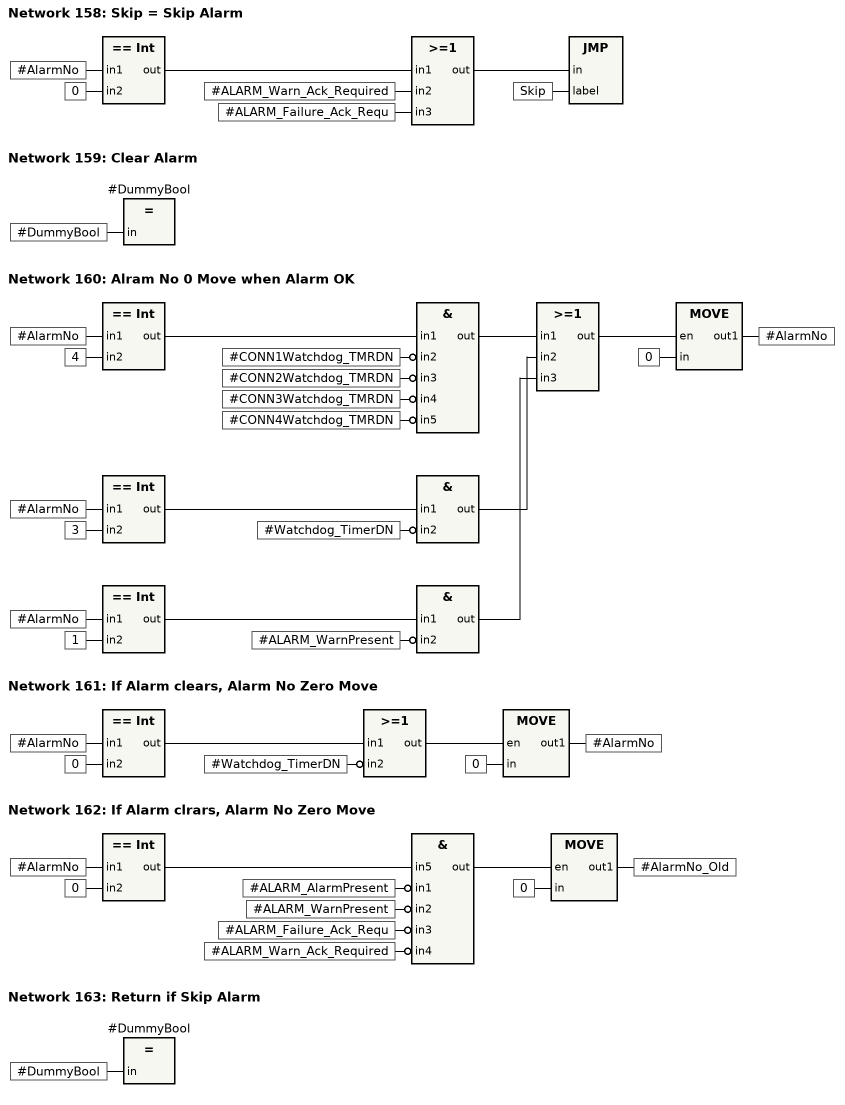
   IF (#AlarmNo = 0) OR #ALARM_Warn_Ack_Required OR #ALARM_Failure_Ack_Requ THEN GOTO Skip; END_IF;
END_REGION

REGION Network 159: Clear Alarm
   // >>>>>>>Clear Alarm>>>>>>>
   Clr:
   #DummyBool := #DummyBool;
END_REGION

REGION Network 160: Alram No 0 Move when Alarm OK
   IF ((#AlarmNo = 4) AND NOT #CONN1Watchdog_TMRDN AND NOT #CONN2Watchdog_TMRDN AND NOT #CONN3Watchdog_TMRDN AND NOT #CONN4Watchdog_TMRDN) OR ((#AlarmNo = 3) AND NOT #Watchdog_TimerDN) OR ((#AlarmNo = 1) AND NOT #ALARM_WarnPresent) THEN
       #AlarmNo := 0;
   END_IF;
END_REGION

REGION Network 161: If Alarm clears, Alarm No Zero Move
   IF (#AlarmNo = 0) OR NOT #Watchdog_TimerDN THEN #AlarmNo := 0; END_IF;
END_REGION

REGION Network 162: If Alarm clrars, Alarm No Zero Move
   IF (#AlarmNo = 0) AND NOT #ALARM_AlarmPresent AND NOT #ALARM_WarnPresent AND NOT #ALARM_Failure_Ack_Requ AND NOT #ALARM_Warn_Ack_Required THEN
       #AlarmNo_Old := 0;
   END_IF;
END_REGION

REGION Network 163: Return if Skip Alarm
   Skip:
   #DummyBool := #DummyBool;
END_REGION

REGION Network 164: Bit 16-19: Mode
   // 0 = Auto
   // 1= Single Start
   // 2 = Manual
   // 3= Local
   // 4= Test Mode
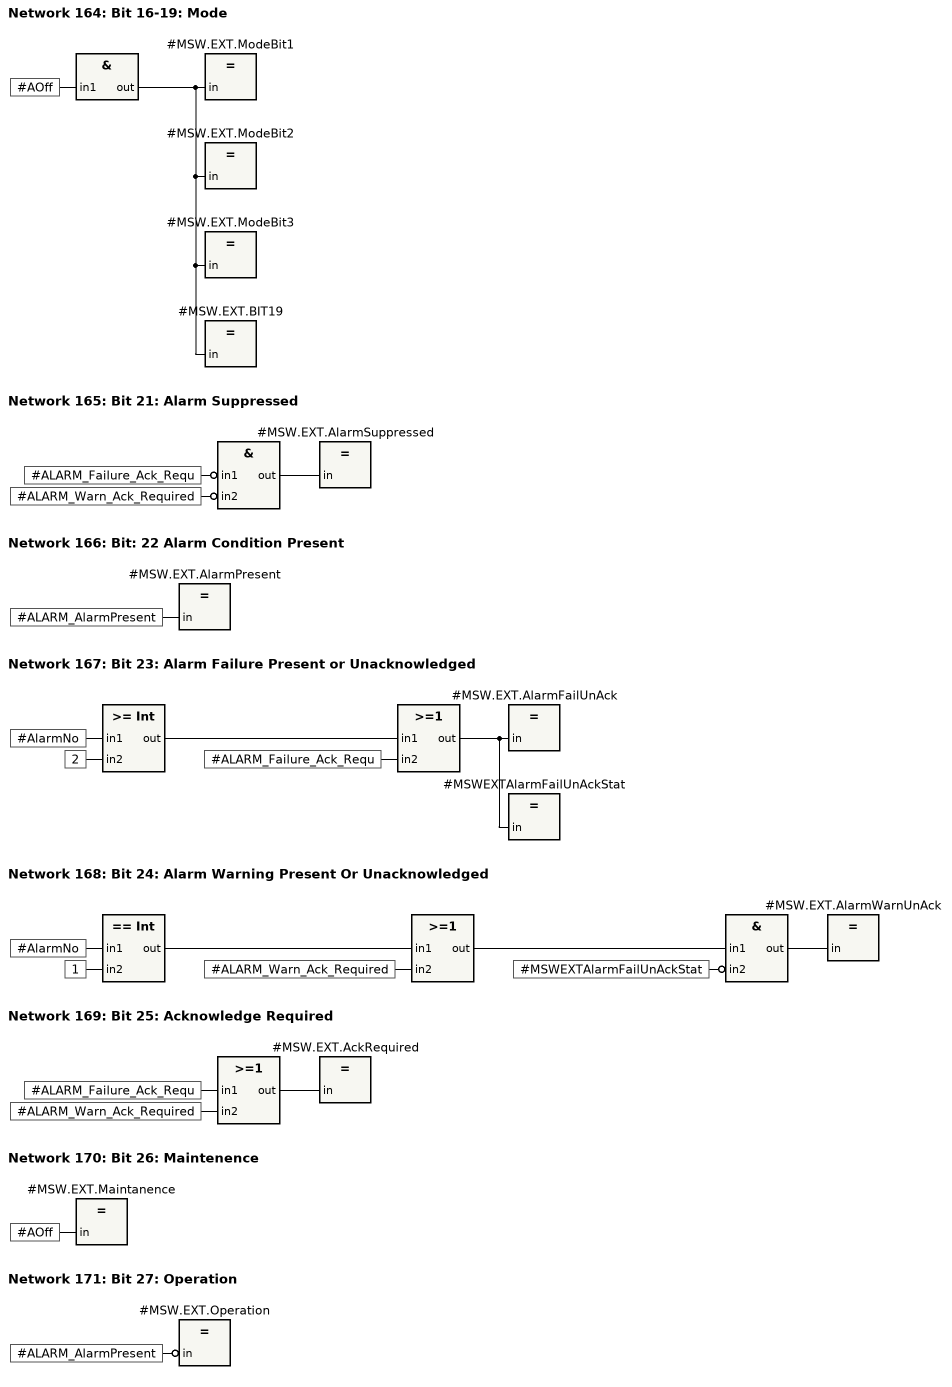
   #MSW.EXT.ModeBit1 := #AOff;
   #MSW.EXT.ModeBit2 := #AOff;
   #MSW.EXT.ModeBit3 := #AOff;
   #MSW.EXT.BIT19 := #AOff;
END_REGION

REGION Network 165: Bit 21: Alarm Suppressed
   #MSW.EXT.AlarmSuppressed := NOT #ALARM_Failure_Ack_Requ AND NOT #ALARM_Warn_Ack_Required;
END_REGION

REGION Network 166: Bit: 22 Alarm Condition Present
   #MSW.EXT.AlarmPresent := #ALARM_AlarmPresent;
END_REGION

REGION Network 167: Bit 23: Alarm Failure Present or Unacknowledged
   #MSW.EXT.AlarmFailUnAck := (#AlarmNo >= 2) OR #ALARM_Failure_Ack_Requ;
   #MSWEXTAlarmFailUnAckStat := #MSW.EXT.AlarmFailUnAck;
END_REGION

REGION Network 168: Bit 24: Alarm Warning Present Or Unacknowledged
   #MSW.EXT.AlarmWarnUnAck := ((#AlarmNo = 1) OR #ALARM_Warn_Ack_Required) AND NOT #MSWEXTAlarmFailUnAckStat;
END_REGION

REGION Network 169: Bit 25: Acknowledge Required
   #MSW.EXT.AckRequired := #ALARM_Failure_Ack_Requ OR #ALARM_Warn_Ack_Required;
END_REGION

REGION Network 170: Bit 26: Maintenence
   #MSW.EXT.Maintanence := #AOff;
END_REGION

REGION Network 171: Bit 27: Operation
   #MSW.EXT.Operation := NOT #ALARM_AlarmPresent;
END_REGION

REGION Network 172: Bit 28: Forced
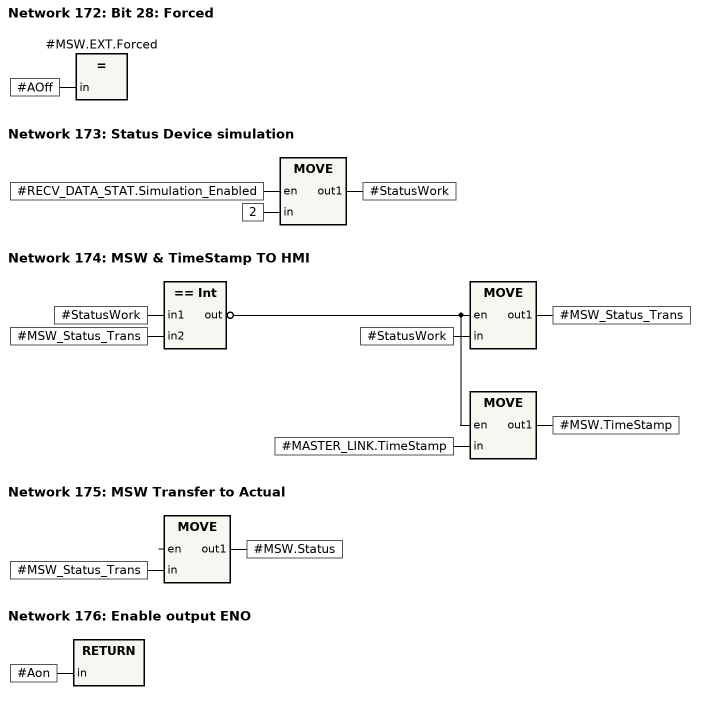
   #MSW.EXT.Forced := #AOff;
END_REGION

REGION Network 173: Status Device simulation
   IF #RECV_DATA_STAT.Simulation_Enabled THEN #StatusWork := 2; END_IF;
END_REGION

REGION Network 174: MSW & TimeStamp TO HMI
   #_w1 := NOT (#StatusWork = #MSW_Status_Trans);
   IF #_w1 THEN
       #MSW_Status_Trans := #StatusWork;
       #MSW.TimeStamp := #MASTER_LINK.TimeStamp;
   END_IF;
END_REGION

REGION Network 175: MSW Transfer to Actual
   #MSW.Status := #MSW_Status_Trans;
END_REGION

REGION Network 176: Enable output ENO
   IF #Aon THEN
       ENO := TRUE;
       RETURN;
   END_IF;
END_REGION
END_FUNCTION_BLOCK

FUNCTION_BLOCK "ACESYS_ISO_On_TCP_TSAP"   // FB228, FBD
TITLE = ACESYS V8.0 - Build 001 - ACESYS_ISO_On_TCP_TSAP
{ S7_Optimized_Access := 'FALSE' }
AUTHOR : FLSMIDTH
FAMILY : ACESYS
NAME : ISO_ON_TCP_TSAP
VERSION : 8.0
// Reference Block of ACESYS_SEND_RECV
   VAR_INPUT
      From_TCON_FC : Struct
         Connection_ID : Word;   // Valid from W#16#0001 to W#16#0FFF
         Connection_DEV_ID : Byte;   // B#16#01-IM151,#02-CPU31x,#03-S7319,#05-400CPU0,#15-400CPU1,#00-CP,10-CP(CPU1)
         Connection_ACT : Bool;   // ACTIVE=1; PASSIVE=0
         Connection_IP_ADDR1 : Int;   // Connection IP Address 1
         Connection_IP_ADDR2 : Int;   // Connection IP Address 2
         Connection_IP_ADDR3 : Int;   // Connection IP Address 3
         Connection_IP_ADDR4 : Int;   // Connection IP Address 4
         Connection_LOC_RS : Byte;   // Connection Local Rack/Slot
         Connection_CP_RS : Byte;   // Connection CP Rack/Slot
         Connection_REM_RS : Byte;   // Connection Remote Rack/Slot
         Connection_CONFIG_NO : Byte;   // B#16#01-CPU0NetA,#02CPU0NetB,#03CPU1NetA,#04CPU1NetB
      END_STRUCT;
   END_VAR
   VAR_OUTPUT
      TCON_PARM : TCON_IP_RFC;
   END_VAR
   VAR
      BlockInfo : Struct
         Ace_Version : Int;   // Acesys Block Version Number
         Ace_BuildNo : Int;   // Acesys Block Build Number
         DB_Number : Int;   // Block Instance DB Number
      END_STRUCT;
      SPECIFIED : Bool;
      DummyString : String[16];
      Connection_ID_Old : Word;
      Conn_String : String[16];
      TSAP16 : String[16];
      ID AT TSAP16 : Array[1..18] of Byte;
      Conn_EXT_HWID : GEOADDR;
   END_VAR
   VAR_TEMP
      Aon : Bool;
      DummyBool : Bool;
      DummyDWord : DWord;
      DummyInt : Int;
      DummyDInt : DInt;
      RET : Int;
      LOC_LEN : Int;
      REM_LEN : Int;
      TMP_INT : Int;
      LOC_RS : Int;
      TMP_RS : Int;
      TMP_DEV : Int;
      UDT_Length : Int;
      t_Zero : Int;
      Sample : Array[1..16] of Byte;
      b_Zero : Array[0..1] of Byte;
   END_VAR
   VAR_TEMP   // added for the SCL form of the ladder/FBD networks
      _w1 : Bool;
      _w2 : Bool;
      _w3 : Bool;
   END_VAR
BEGIN

REGION Network 1: Acesys Send Function Block based on Open Communication standard
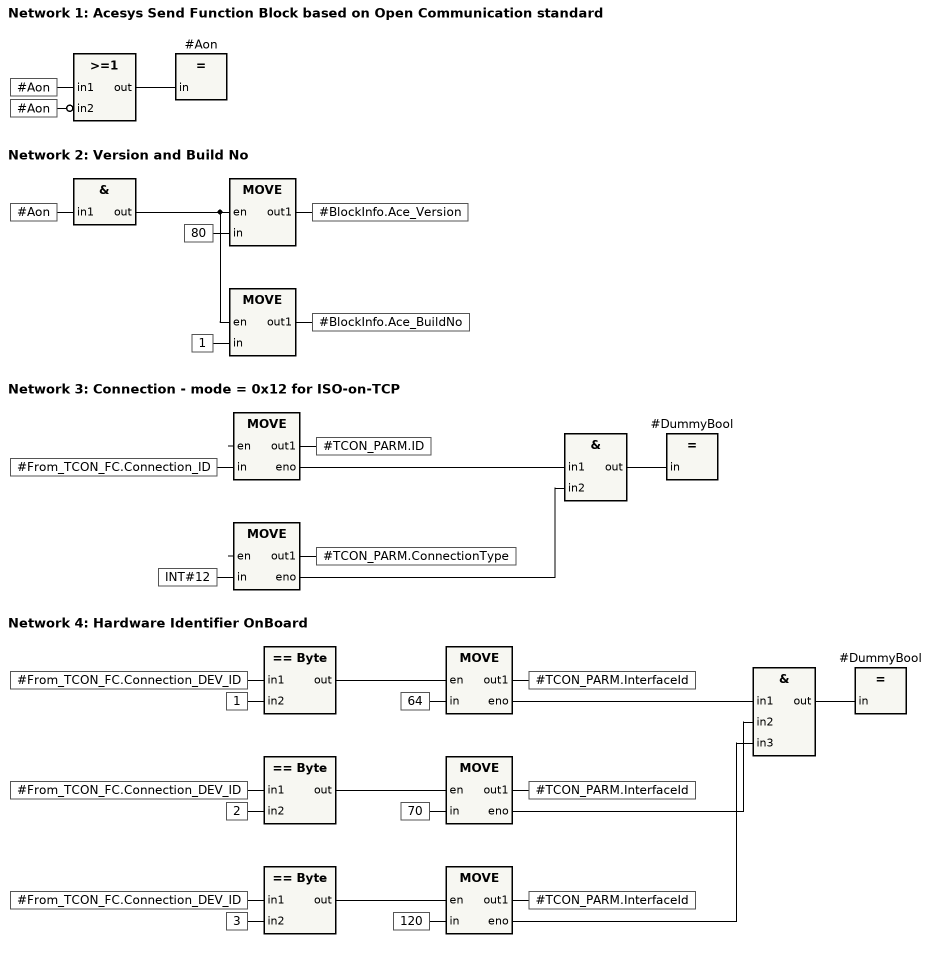
   #Aon := #Aon OR NOT #Aon;
END_REGION

REGION Network 2: Version and Build No
   IF #Aon THEN
       #BlockInfo.Ace_Version := 80;
       #BlockInfo.Ace_BuildNo := 1;
   END_IF;
END_REGION

REGION Network 3: Connection - mode = 0x12 for ISO-on-TCP
   // ENO of a box is taken as its EN; it also drops when the box reports an error
   #TCON_PARM.ID := #From_TCON_FC.Connection_ID;
   #TCON_PARM.ConnectionType := INT#12;
   #DummyBool := TRUE;
END_REGION

REGION Network 4: Hardware Identifier OnBoard
   #_w1 := #From_TCON_FC.Connection_DEV_ID = 1;
   IF #_w1 THEN #TCON_PARM.InterfaceId := 64; END_IF;
   #_w2 := #From_TCON_FC.Connection_DEV_ID = 2;
   IF #_w2 THEN #TCON_PARM.InterfaceId := 70; END_IF;
   #_w3 := #From_TCON_FC.Connection_DEV_ID = 3;
   IF #_w3 THEN #TCON_PARM.InterfaceId := 120; END_IF;
   #DummyBool := #_w1 AND #_w2 AND #_w3;
END_REGION

REGION Network 5: Hardware Identifier External
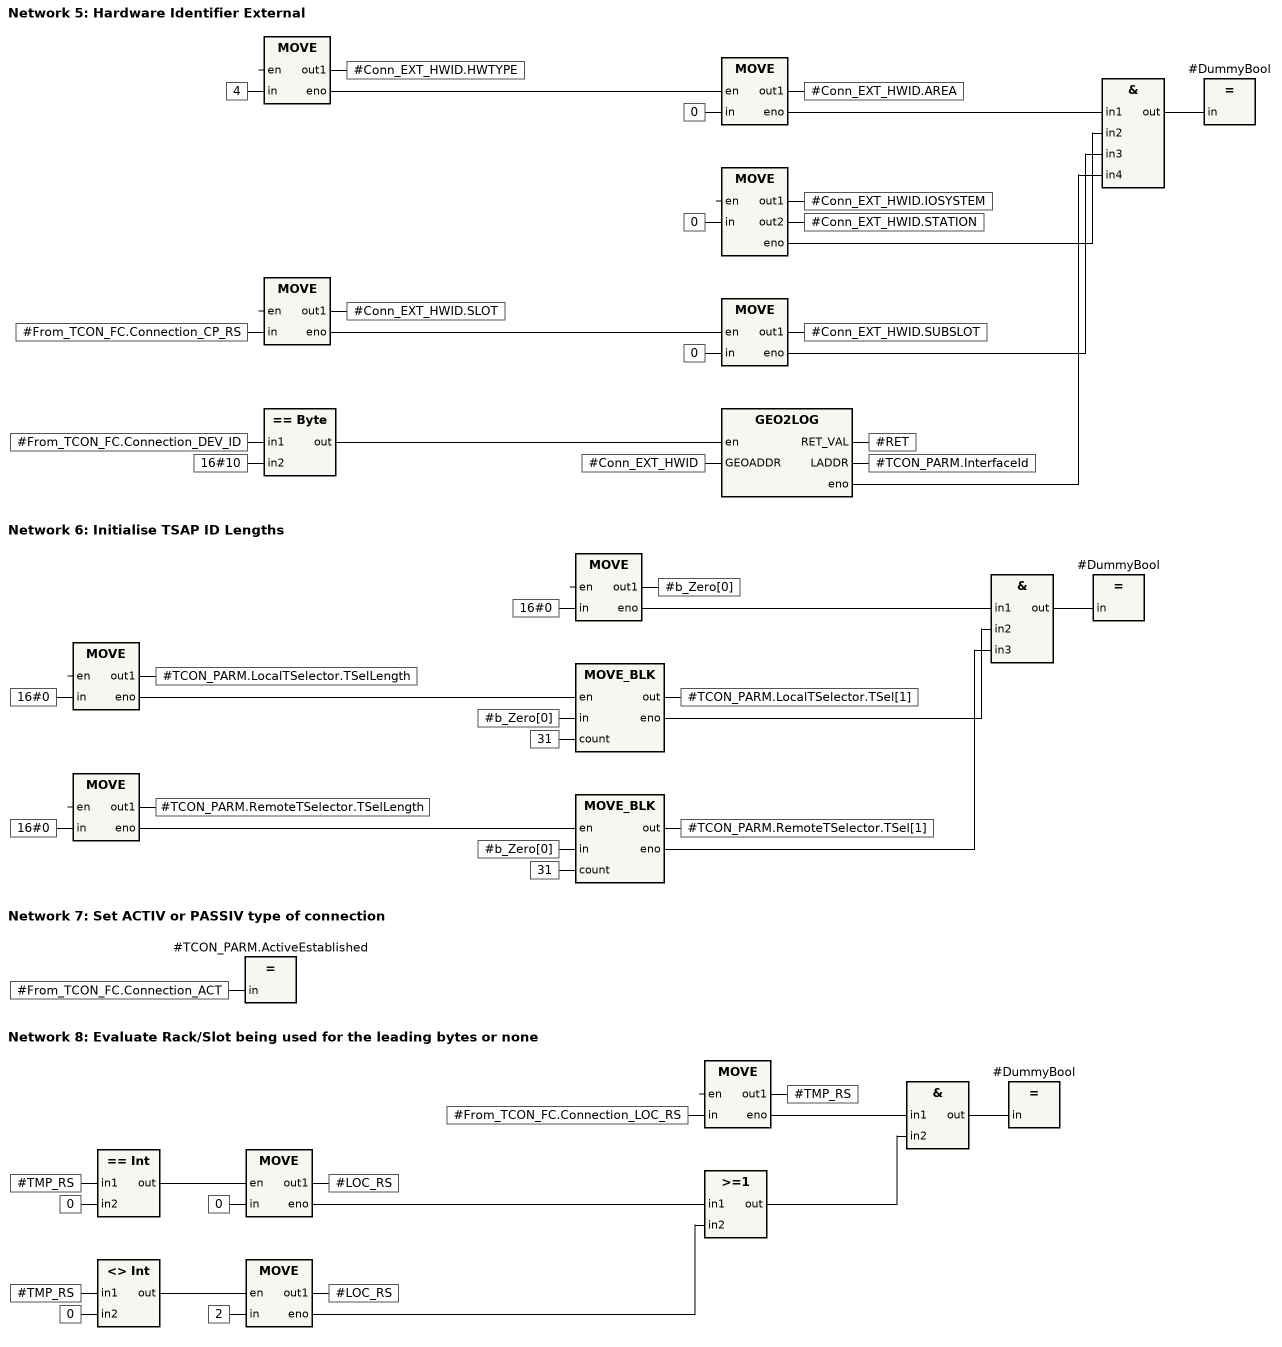
   // ENO of a box is taken as its EN; it also drops when the box reports an error
   #Conn_EXT_HWID.HWTYPE := 4;
   #Conn_EXT_HWID.AREA := 0;
   #Conn_EXT_HWID.IOSYSTEM := 0;
   #Conn_EXT_HWID.STATION := 0;
   #Conn_EXT_HWID.SLOT := #From_TCON_FC.Connection_CP_RS;
   #Conn_EXT_HWID.SUBSLOT := 0;
   #_w1 := #From_TCON_FC.Connection_DEV_ID = 16#10;
   IF #_w1 THEN #RET := GEO2LOG(GEOADDR := #Conn_EXT_HWID, LADDR => #TCON_PARM.InterfaceId); END_IF;
   #DummyBool := #_w1;
END_REGION

REGION Network 6: Initialise TSAP ID Lengths
   #b_Zero[0] := 16#0;
   #TCON_PARM.LocalTSelector.TSelLength := 16#0;
   MOVE_BLK(IN := #b_Zero[0], COUNT := 31, OUT => #TCON_PARM.LocalTSelector.TSel[1]);
   #TCON_PARM.RemoteTSelector.TSelLength := 16#0;
   MOVE_BLK(IN := #b_Zero[0], COUNT := 31, OUT => #TCON_PARM.RemoteTSelector.TSel[1]);
   #DummyBool := TRUE;
END_REGION

REGION Network 7: Set ACTIV or PASSIV type of connection
   // Receive Block Always Pasive
   #TCON_PARM.ActiveEstablished := #From_TCON_FC.Connection_ACT;
END_REGION

REGION Network 8: Evaluate Rack/Slot being used for the leading bytes or none
   // 1) If R/S = 0 ---> no leading bytes are requested.
   // 2) If R/S # 0 ---> two leading bytes are required.
   // ENO of a box is taken as its EN; it also drops when the box reports an error
   #TMP_RS := #From_TCON_FC.Connection_LOC_RS;
   #_w1 := #TMP_RS = 0;
   IF #_w1 THEN #LOC_RS := 0; END_IF;
   #_w2 := #TMP_RS <> 0;
   IF #_w2 THEN #LOC_RS := 2; END_IF;
   #DummyBool := #_w1 OR #_w2;
END_REGION

REGION Network 9: Check if ID is Changed
   // #MASTER_LINK.FIRST_SCAN - Removed
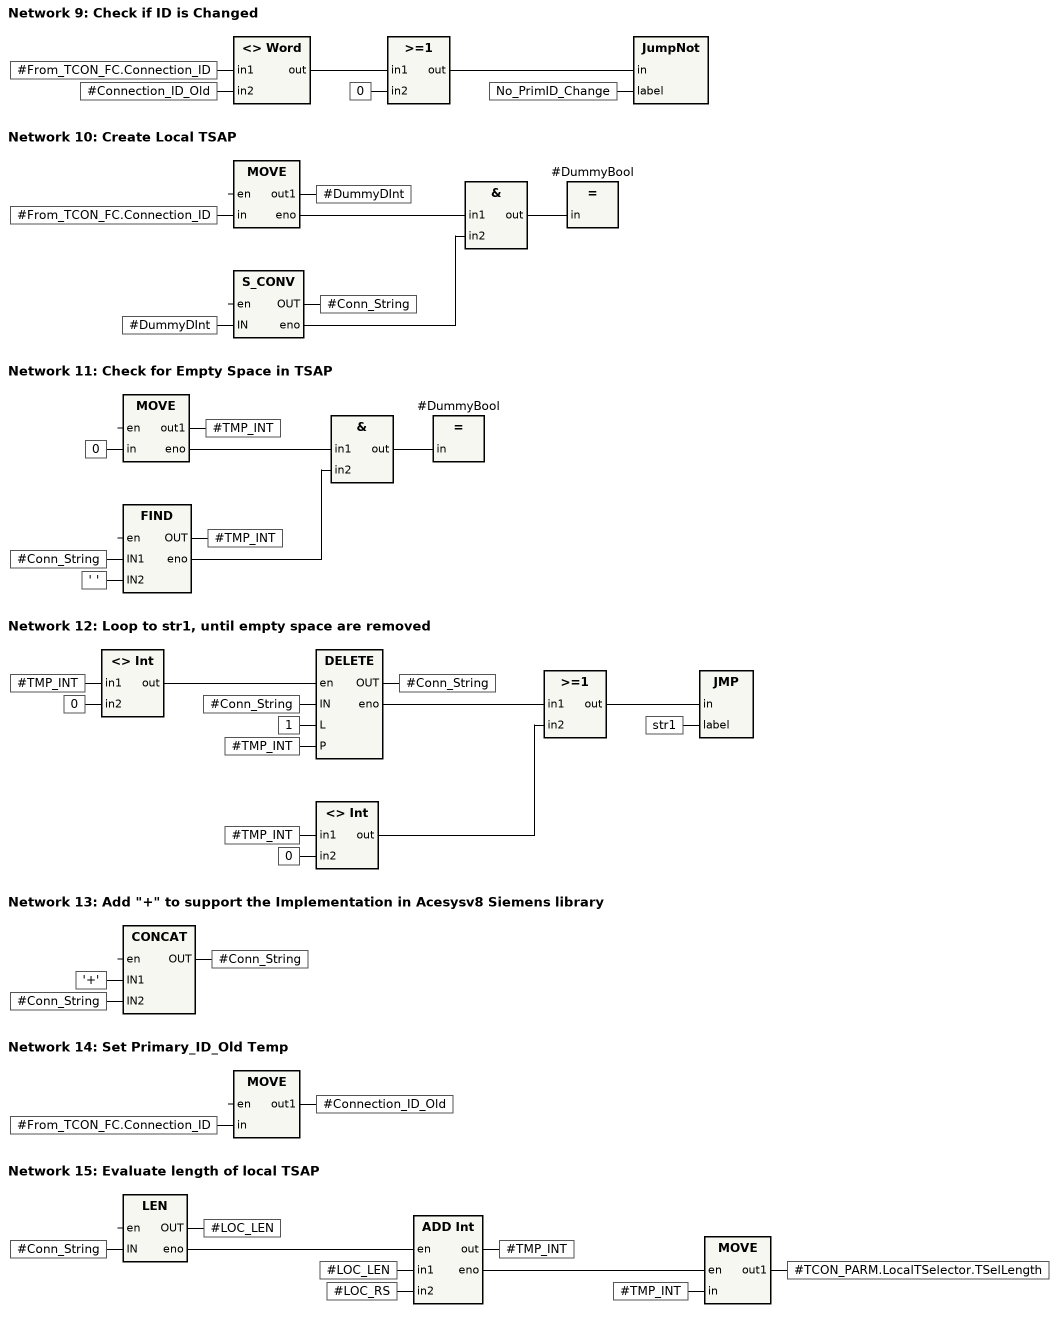
   // no SCL statement known for JumpNot: written as a call
   JumpNot(in := (#From_TCON_FC.Connection_ID <> #Connection_ID_Old) OR 0, label := No_PrimID_Change);
END_REGION

REGION Network 10: Create Local TSAP
   // Local TSAP = ID_Number
   // ENO of a box is taken as its EN; it also drops when the box reports an error
   #DummyDInt := #From_TCON_FC.Connection_ID;
   #Conn_String := S_CONV(IN := #DummyDInt);
   #DummyBool := TRUE;
END_REGION

REGION Network 11: Check for Empty Space in TSAP
   str1:
   #TMP_INT := 0;
   #TMP_INT := FIND(IN1 := #Conn_String, IN2 := ' ');
   #DummyBool := TRUE;
END_REGION

REGION Network 12: Loop to str1, until empty space are removed
   #_w1 := #TMP_INT <> 0;
   IF #_w1 THEN #Conn_String := DELETE(IN := #Conn_String, L := 1, P := #TMP_INT); END_IF;
   IF #_w1 OR (#TMP_INT <> 0) THEN GOTO str1; END_IF;
END_REGION

REGION Network 13: Add "+" to support the Implementation in Acesysv8 Siemens library
   #Conn_String := CONCAT(IN1 := '+', IN2 := #Conn_String);
END_REGION

REGION Network 14: Set Primary_ID_Old Temp
   No_PrimID_Change:
   #Connection_ID_Old := #From_TCON_FC.Connection_ID;
END_REGION

REGION Network 15: Evaluate length of local TSAP
   // #TSAP.LOC_TSAP
   // ENO of a box is taken as its EN; it also drops when the box reports an error
   #LOC_LEN := LEN(IN := #Conn_String);
   #TMP_INT := #LOC_LEN + #LOC_RS;
   #TCON_PARM.LocalTSelector.TSelLength := #TMP_INT;
END_REGION

REGION Network 16: copy local TSAP String to TSAP16 String!
   // #TSAP.LOC_TSAP
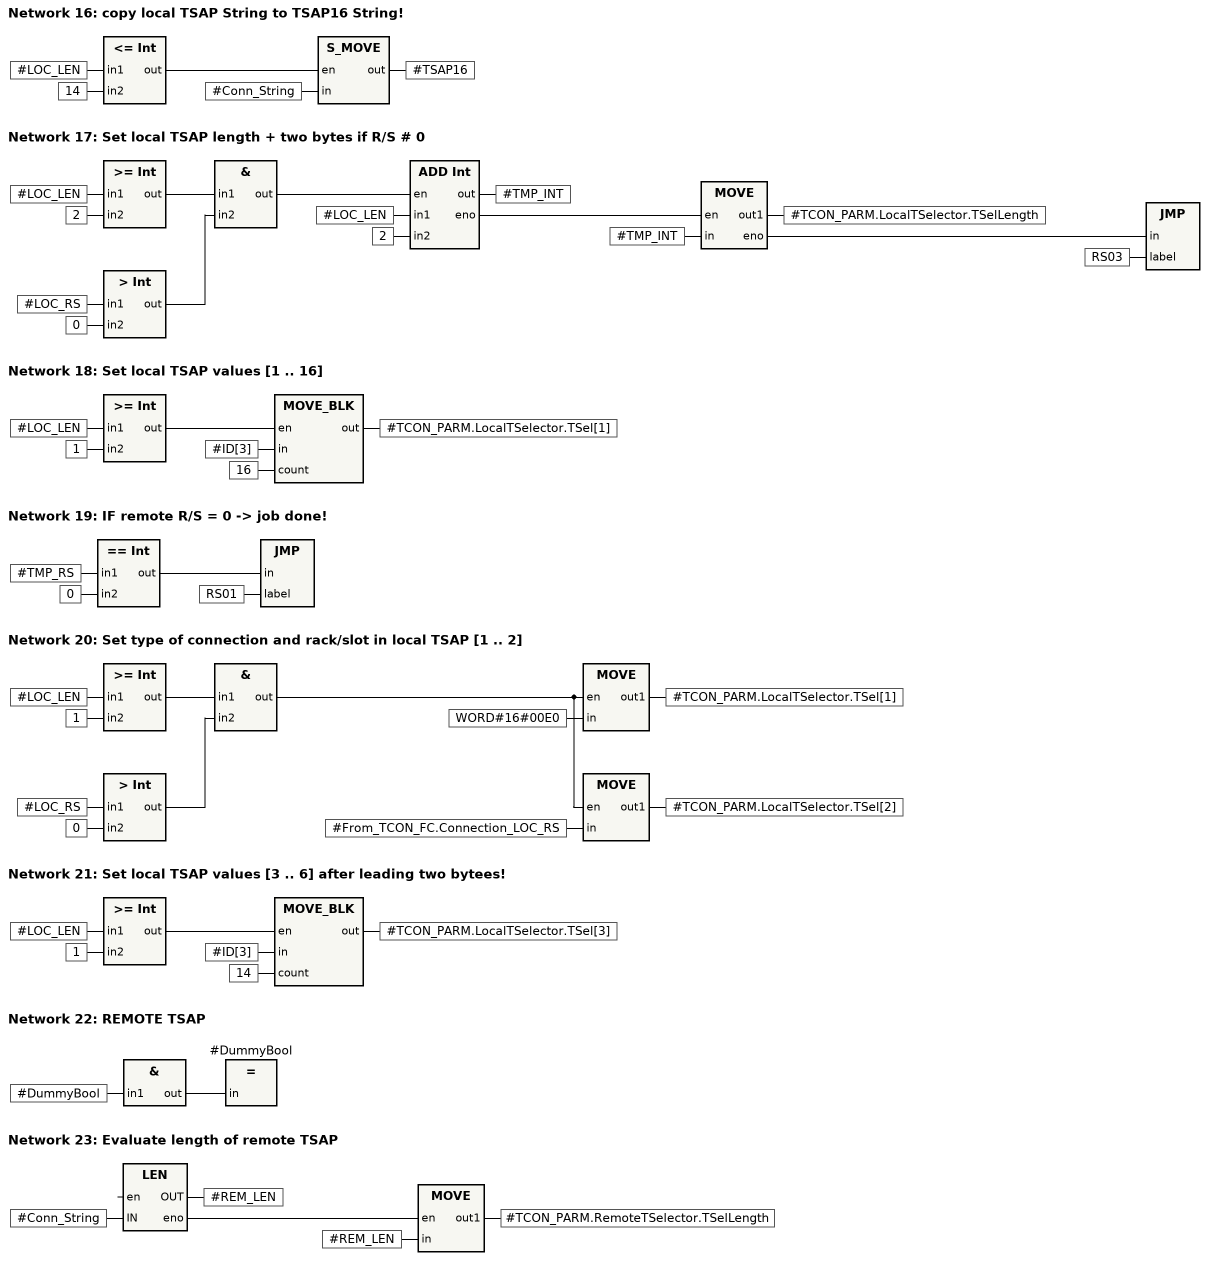
   IF #LOC_LEN <= 14 THEN #TSAP16 := #Conn_String; END_IF;
END_REGION

REGION Network 17: Set local TSAP length + two bytes if R/S # 0
   // ENO of a box is taken as its EN; it also drops when the box reports an error
   #_w1 := (#LOC_LEN >= 2) AND (#LOC_RS > 0);
   IF #_w1 THEN
       #TMP_INT := #LOC_LEN + 2;
       #TCON_PARM.LocalTSelector.TSelLength := #TMP_INT;
       GOTO RS03;
   END_IF;
END_REGION

REGION Network 18: Set local TSAP values [1 .. 16]
   // Fill in the entire local TSAP (without leading bytes)
   IF #LOC_LEN >= 1 THEN
       MOVE_BLK(IN := #ID[3], COUNT := 16, OUT => #TCON_PARM.LocalTSelector.TSel[1]);
   END_IF;
END_REGION

REGION Network 19: IF remote R/S = 0 -> job done!
   IF #TMP_RS = 0 THEN GOTO RS01; END_IF;
END_REGION

REGION Network 20: Set type of connection and rack/slot in local TSAP [1 .. 2]
   // B#16#E0 -> type of connection 
   // B#16#02 -> rack/slot of CPU
   RS03:
   IF (#LOC_LEN >= 1) AND (#LOC_RS > 0) THEN
       #TCON_PARM.LocalTSelector.TSel[1] := WORD#16#00E0;
       #TCON_PARM.LocalTSelector.TSel[2] := #From_TCON_FC.Connection_LOC_RS;
   END_IF;
END_REGION

REGION Network 21: Set local TSAP values [3 .. 6] after leading two bytees!
   IF #LOC_LEN >= 1 THEN
       MOVE_BLK(IN := #ID[3], COUNT := 14, OUT => #TCON_PARM.LocalTSelector.TSel[3]);
   END_IF;
END_REGION

REGION Network 22: REMOTE TSAP
   RS01:
   #DummyBool := #DummyBool;
END_REGION

REGION Network 23: Evaluate length of remote TSAP
   // Remote TSAP = Local TSAP (DummyString1)
   #REM_LEN := LEN(IN := #Conn_String);
   #TCON_PARM.RemoteTSelector.TSelLength := #REM_LEN;
END_REGION

REGION Network 24: copy remote TSAP String to TSAP16 String!
   // Remote TSAP = Local TSAP (DummyString)
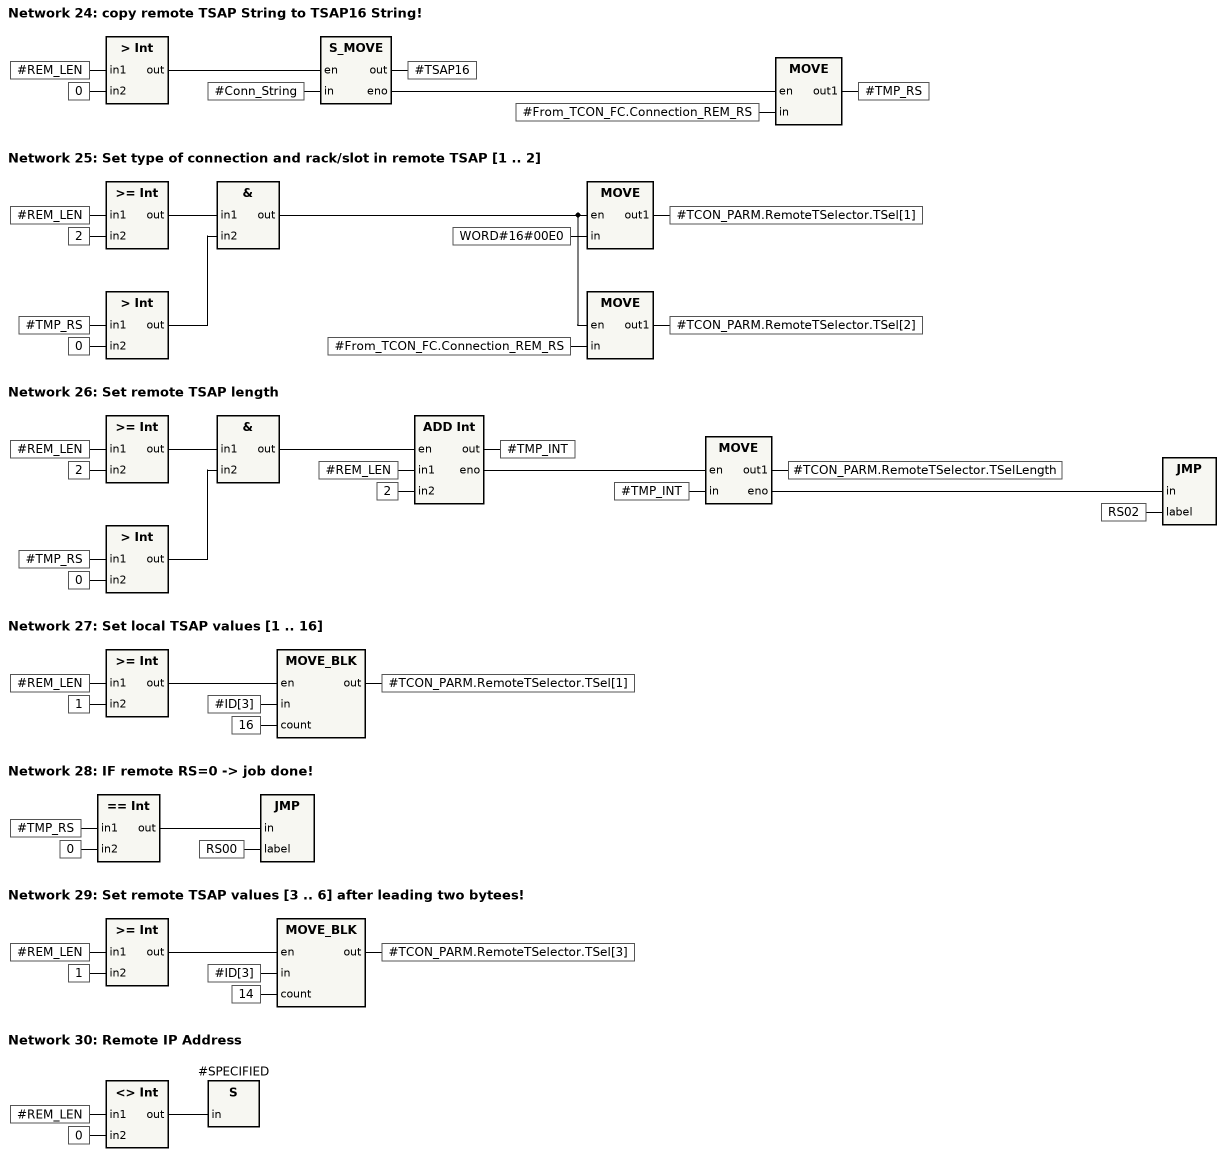
   IF #REM_LEN > 0 THEN
       #TSAP16 := #Conn_String;
       #TMP_RS := #From_TCON_FC.Connection_REM_RS;
   END_IF;
END_REGION

REGION Network 25: Set type of connection and rack/slot in remote TSAP [1 .. 2]
   // B#16#E0 -> type of connection 
   // B#16#02 -> rack/slot of CPU
   IF (#REM_LEN >= 2) AND (#TMP_RS > 0) THEN
       #TCON_PARM.RemoteTSelector.TSel[1] := WORD#16#00E0;
       #TCON_PARM.RemoteTSelector.TSel[2] := #From_TCON_FC.Connection_REM_RS;
   END_IF;
END_REGION

REGION Network 26: Set remote TSAP length
   // ENO of a box is taken as its EN; it also drops when the box reports an error
   #_w1 := (#REM_LEN >= 2) AND (#TMP_RS > 0);
   IF #_w1 THEN
       #TMP_INT := #REM_LEN + 2;
       #TCON_PARM.RemoteTSelector.TSelLength := #TMP_INT;
       GOTO RS02;
   END_IF;
END_REGION

REGION Network 27: Set local TSAP values [1 .. 16]
   // Fill in the entire local TSAP (without leading bytes)
   IF #REM_LEN >= 1 THEN
       MOVE_BLK(IN := #ID[3], COUNT := 16, OUT => #TCON_PARM.RemoteTSelector.TSel[1]);
   END_IF;
END_REGION

REGION Network 28: IF remote RS=0 -> job done!
   IF #TMP_RS = 0 THEN GOTO RS00; END_IF;
END_REGION

REGION Network 29: Set remote TSAP values [3 .. 6] after leading two bytees!
   RS02:
   IF #REM_LEN >= 1 THEN
       MOVE_BLK(IN := #ID[3], COUNT := 14, OUT => #TCON_PARM.RemoteTSelector.TSel[3]);
   END_IF;
END_REGION

REGION Network 30: Remote IP Address
   // Set length of the IP address if full-specified only !
   RS00:
   IF #REM_LEN <> 0 THEN #SPECIFIED := TRUE; END_IF;
END_REGION

REGION Network 31: Set not length of the IP address if unspecified !!!!
   // The remote IP address must be zero if
   // 1) remote TSAP is unspecified, or
   // 2) IP address is set up with zero!
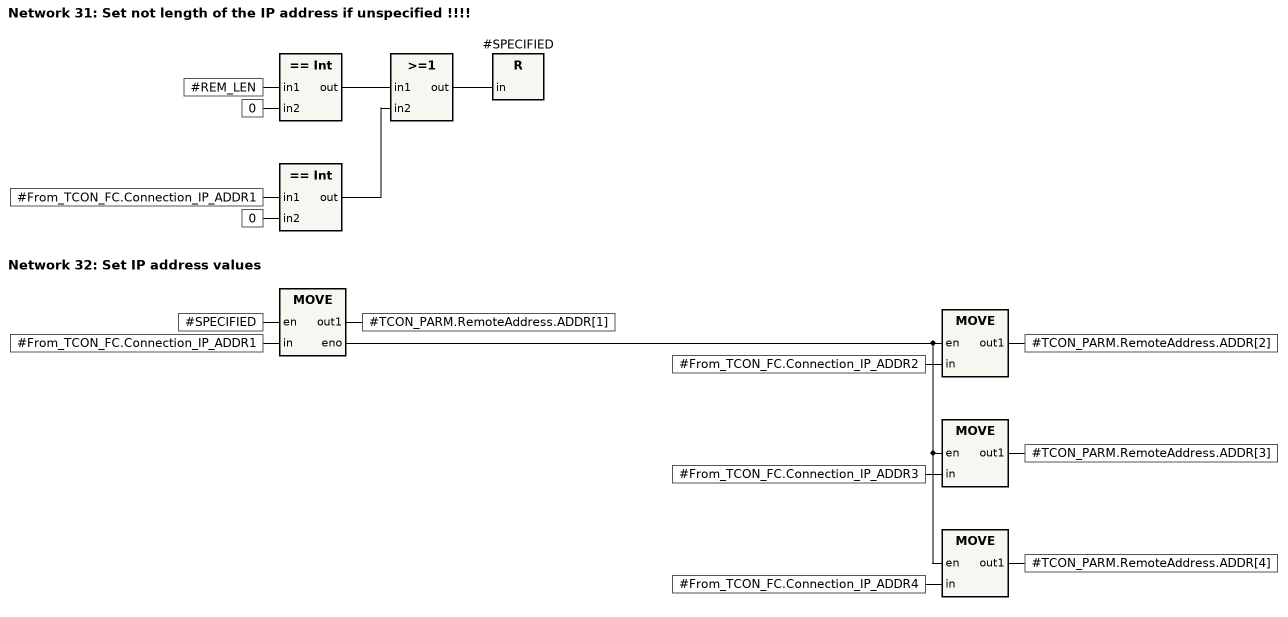
   IF (#REM_LEN = 0) OR (#From_TCON_FC.Connection_IP_ADDR1 = 0) THEN #SPECIFIED := FALSE; END_IF;
END_REGION

REGION Network 32: Set IP address values
   // ENO of a box is taken as its EN; it also drops when the box reports an error
   IF #SPECIFIED THEN
       #TCON_PARM.RemoteAddress.ADDR[1] := #From_TCON_FC.Connection_IP_ADDR1;
       #TCON_PARM.RemoteAddress.ADDR[2] := #From_TCON_FC.Connection_IP_ADDR2;
       #TCON_PARM.RemoteAddress.ADDR[3] := #From_TCON_FC.Connection_IP_ADDR3;
       #TCON_PARM.RemoteAddress.ADDR[4] := #From_TCON_FC.Connection_IP_ADDR4;
   END_IF;
END_REGION
END_FUNCTION_BLOCK

FUNCTION_BLOCK "ACESYS_PLC_DIAGV2"   // FB229, SCL
{ S7_Optimized_Access := 'FALSE' }
VERSION : 0.1
   VAR_INPUT
      HSBY_EN : Bool;   // Future Use
      OB33_ScanTime_In : Int;
      OB35_ScanTime_In : Int;
      CPU_Type : Int;   // Valid NO: "1200", "1500"
      Master_Link : "ACESYS_MASTER_LINK";
   END_VAR
   VAR_OUTPUT
      CPU_OK : Bool;   // CPU Status OK
      Type_Fault : Bool;   // CPU Type Fault
      CPUClock_Sec : USInt;
      CPUClock_Min : USInt;
      CPUClock_Hour : USInt;
      CPUClock_Day : USInt;
      CPUClock_Month : USInt;
      CPUClock_Year : UInt;
      OB01_ScanTime : Int;
      OB33_ScanTime : Int;
      OB35_ScanTime : Int;
      Memory_Total : DInt;
      Memory_Used : DInt;
      Mem_UsePercentage : Real;
      MSW : "ACESYS_HMI_STAT_32T";
   END_VAR
   VAR
      BlockInfo : Struct
         Ace_Version : Int;   // Acesys Block Version Number
         Ace_BuildNo : Int;   // Acesys Block Build Number
         DB_Number : Int;   // Block Instance DB Number
      END_STRUCT;
      FP_CMD : Struct   // Faceplate Commands
         Spare_08 : Bool;   // Bit8
         Spare_09 : Bool;   // Bit9
         Spare_10 : Bool;   // Bit10
         Spare_11 : Bool;   // Bit11
         Spare_12 : Bool;   // Bit12
         Spare_13 : Bool;   // Bit13
         Spare_14 : Bool;   // Bit14
         AckAlarm : Bool;   // Alarm Acknowledge
         Spare_00 : Bool;   // Bit0
         Spare_01 : Bool;   // Bit1
         Spare_02 : Bool;   // Bit2
         Spare_03 : Bool;   // Bit3
         Spare_04 : Bool;   // Bit4
         Spare_05 : Bool;   // Bit5
         Spare_06 : Bool;   // Bit6
         Spare_07 : Bool;   // Bit7
      END_STRUCT;
      FP_DIM : Struct
         Spare16 : Bool;
         Spare15 : Bool;
         Spare14 : Bool;
         Spare13 : Bool;
         Spare12 : Bool;
         Spare11 : Bool;
         Spare10 : Bool;
         Spare09 : Bool;
         Spare08 : Bool;
         Spare07 : Bool;
         Spare06 : Bool;
         Spare05 : Bool;
         Spare04 : Bool;
         Spare03 : Bool;
         Spare02 : Bool;
         Spare01 : Bool;
      END_STRUCT;
      FP_SHOW : Struct
         CPU_RUN_IND : Bool;
         Spare20 : Bool;
         Spare19 : Bool;
         Spare18 : Bool;
         Spare17 : Bool;
         Spare16 : Bool;
         Spare15 : Bool;
         Spare14 : Bool;
         Spare13 : Bool;
         Spare12 : Bool;
         Spare11 : Bool;
         CPU_MAINT : Bool;
         CPU_ERROR : Bool;
         OB1_ScanTime : Bool;
         OB33_ScanTime : Bool;
         OB35_ScanTime : Bool;
         Memory_Total : Bool;
         Memory_Used : Bool;
         Memory_Percent : Bool;
         Spare_10 : Bool;
         Spare_09 : Bool;
         Spare_08 : Bool;
         OB33ScanTimeIn : Bool;
         OB35ScanTimeIn : Bool;
         Spare_07 : Bool;
         Spare_06 : Bool;
         Spare_05 : Bool;
         Spare_04 : Bool;
         Spare_03 : Bool;
         Spare_02 : Bool;
         Spare_01 : Bool;
         Spare_00 : Bool;
      END_STRUCT;
      FP_PARM : Struct
         Spare16 : Bool;
         Spare15 : Bool;
         Spare14 : Bool;
         Spare13 : Bool;
         Spare12 : Bool;
         Spare11 : Bool;
         Spare10 : Bool;
         Spare09 : Bool;
         Spare08 : Bool;
         Spare07 : Bool;
         Spare06 : Bool;
         Spare05 : Bool;
         Spare04 : Bool;
         Spare03 : Bool;
         Spare02 : Bool;
         Spare01 : Bool;
      END_STRUCT;
      StatusWork : Int;
      StatusBuilder : Int;
      SFC51_RET_VAL_Spare : Int;
      SFC51_BUSY_Spare : Bool;
      SZL_HEADER_Spare : Struct
         LENGTHDR : Word;
         N_DR : Word;
      END_STRUCT;
      Spare_W8 : Word;   // LED RUN Check
      Spare_W9 : Word;   // LED ERROR Check
      Spare_W10 : Word;   // LED MAINT Check
      Spare_W11 : Word;
      Spare_W12 : Word;
      Spare_W13 : Word;
      Spare_W14 : Word;
      Spare_W15 : Word;
      Record_LED_MAINT : Word;
      Spare_W16 : Word;
      Record_LED_ERROR : Word;
      Spare_W2 : Word;
      Spare_W3 : Word;
      Spare_W4 : Word;
      Spare_W5 : Word;
      Spare_W6 : Word;
      Spare_W7 : Word;
      Spare_W17 : Word;
      AlarmNo : Int;
      AlarmNo_Old : Int;
      ALARM_AlarmPresent : Bool;
      ALARM_Failure_Ack_Requ : Bool;
      CMD_Acknowledge : Bool;   // Internal Acknowledge
      ALARM_SuppresionActiv : Bool;
      Type_1200 : Bool;   // Type 300 Selected
      Type_1500 : Bool;   // Type 400 Selected
      Spare25 : Bool;   // CPU RUN Indicator Flashing=Run, Steady=Stopped/Error
      CPU_RUN_IND : Bool;   // "1" = CPU LED OK
      Spare24 : Bool;   // "1" = CPU LED OK
      Spare23 : Bool;
      Spare22 : Bool;
      Spare21 : Bool;
      Spare20 : Bool;
      Spare19 : Bool;
      Spare18 : Bool;
      Spare17 : Bool;
      CPU_MAINT : Bool;
      Spare16 : Bool;
      CPU_ERROR : Bool;
      Spare14 : Bool;
      Spare13 : Bool;
      Spare12 : Bool;
      Spare11 : Bool;
      Spare10 : Bool;
      Spare9 : Bool;
      Spare8 : Bool;
      Spare7 : Bool;
      Spare6 : Bool;
      Spare5 : Bool;
      Spare4 : Bool;
      Spare3 : Bool;
      Spare2 : Bool;
      Spare1 : Bool;
      BitVar : Bool;
      Ack : Bool;   // Label
      Clear : Bool;
      ALARM_WarnAckRequired : Bool;
      ALARM_WarnPresent : Bool;
      OUT : Struct
         CPU_OK : Bool;
         Type_Fault : Bool;
      END_STRUCT;
      MSW_Status_Trans : Int;
      GetSMCinfo_Instance : GetSMCinfo;
      GetSMCinfo_Instance_1 : GetSMCinfo;
      GET_IM_DATA_Instance : Get_IM_Data;
   END_VAR
   VAR_TEMP
      LED_Record_Word1 : Word;   // LED Record
      LED_Record_Word2 : Word;   // LED Record
      LED_Record_Word3 : Word;   // LED Record
      LED_Record_Word4 : Word;   // LED Record
      LED_Record_Word5 : Word;   // LED Record
      LED_Record_Word6 : Word;   // LED Record
      LED_Record_Word7 : Word;   // LED Record
      LED_Record_Word8 : Word;   // LED Record
      LED_Record_Word9 : Word;   // LED Record
      LED_Record_Word10 : Word;   // LED Record
      AOn : Bool;   // Always On
      AOff : Bool;   // Always Off
      dummybool : Bool;
      Status_Add : Int;
      AnyPtr : ANY;
      AnyStruct AT AnyPtr : Struct
         S7_ID : Byte;
         Mem_ID : Byte;
         NumberOfElements : Int;
         DB_Number : Word;
         BitPointer : DWord;
      END_STRUCT;
      DummyInt : Int;
      SystemTimeRead : DTL;
      DummyWord : Word;
      DummyDint : DInt;
      DummyReal : Real;
      DummyReal1 : Real;
      DummyUDint : UDInt;
      DATA : Struct
         Manufacturer_ID : UInt;
         Order_ID : String[20];
         Serial_Number : String[20];
         Hardware_Revision : UInt;
         Software_Revision : Struct
            "Type" : Char;
            Functional : USInt;
            Bugfix : USInt;
            Internal : USInt;
         END_STRUCT;
         Revision_Counter : UInt;
         Profile_ID : UInt;
         Profile_Specific_Type : UInt;
         IM_Version : Word;
         IM_Supported : Word;
      END_STRUCT;
      Software_RevisionV1 : Int;
      Software_RevisionV2 : Int;
      Software_RevisionV3 : Int;
   END_VAR
BEGIN
   (* ----------------------------------------------------------------- ACESYS_PLC_DIAGV2  -------------------------------------------------------------*)
   (* ACESYS V8.0 - Build 001 - PLC HW DiagnosticV2 *)
   (* ----------------------------------------------------------------- Block Information -------------------------------------------------------------*)
   (* Version AND Build No *)
   #BlockInfo.Ace_Version := 80;
   #BlockInfo.Ace_BuildNo := 1;

   (* Always On *)
   #AOn := TRUE;
   #AOff := False;
   (* INSTANCE DB Number TO Faceplate *)
   #AnyPtr := #BitVar;
   #BlockInfo.DB_Number := WORD_TO_INT(#AnyStruct.DB_Number);

   (* Automatic Dep_CMD when use OF block interface*)
   #CMD_Acknowledge := #FP_CMD.AckAlarm;
   #FP_CMD.AckAlarm := 0;


   (* Initialize Value*)
   #ALARM_SuppresionActiv := #AOff;
   (* ----------------------------------------------------------------- Type Fault -------------------------------------------------------------*)
   (* Selected CPU Type *)
   IF #CPU_Type = 1500 THEN
       #Type_1500 := TRUE;
   ELSE
       #Type_1500 := False;
   END_IF;

   (* No Type selected *)
   IF NOT #Type_1500 THEN
       #OUT.Type_Fault := TRUE;
   ELSE
       #OUT.Type_Fault := False;
   END_IF;
   (* ----------------------------------------------------------------- Set Show Parameter -------------------------------------------------------------*)
   #FP_SHOW.CPU_RUN_IND := #AOn;
   #FP_SHOW.CPU_MAINT := #AOn;
   #FP_SHOW.CPU_ERROR := #AOn;
   #FP_SHOW.OB1_ScanTime := #AOn;
   #FP_SHOW.OB33_ScanTime := #AOn;
   #FP_SHOW.OB35_ScanTime := #AOn;
   #FP_SHOW.Memory_Total := #AOn;
   #FP_SHOW.Memory_Used := #AOn;
   #FP_SHOW.Memory_Percent := #AOn;
   #FP_SHOW.OB33ScanTimeIn := #AOn;
   #FP_SHOW.OB35ScanTimeIn := #AOn;

   #CPU_RUN_IND := #Master_Link.SEC_Toggle;
   (* ----------------------------------------------------------------- LED Informations -------------------------------------------------------------*)
   (* LED-CPU_ERROR LED Indication *)
   #LED_Record_Word1 := LED(LADDR := 50, LED := 2);
   (* Set Status Flag*)
   #CPU_ERROR := TRUE;
   (*Read ERROR LED Indication*)
   #Record_LED_ERROR := #LED_Record_Word1;
   (*"1" = CPU LED OK*)
   IF #Record_LED_ERROR <> 1 THEN
       #CPU_ERROR := FALSE;
   END_IF;
   (* LED-CPU_MAINT LED Indication *)
   #LED_Record_Word2 := LED(LADDR := 50, LED := 3);
   (* Set Status Flag*)
   #CPU_MAINT := FALSE;
   (*Read Maint LED Indication*)
   #Record_LED_MAINT := #LED_Record_Word2;
   IF #Record_LED_MAINT <> 1 THEN
       #CPU_MAINT := TRUE;
   END_IF;
   (* ----------------------------------------------------------------- CPU RUN Indication -------------------------------------------------------------*)
   (* Run Supervsision Flashing = Run *)
   #Spare25 := #Master_Link.SEC_Toggle;
   (* ----------------------------------------------------------------- CPU Scan Time Information -------------------------------------------------------------*)
   #OB01_ScanTime := #Master_Link.OB1_CycleTime;
   #OB33_ScanTime := #OB33_ScanTime_In;
   #OB35_ScanTime := #OB35_ScanTime_In;
   (* ----------------------------------------------------------------- CPU Clock Read -------------------------------------------------------------*)
   #DummyInt := RD_LOC_T(#SystemTimeRead);
   #CPUClock_Sec := #SystemTimeRead.SECOND;
   #CPUClock_Min := #SystemTimeRead.MINUTE;
   #CPUClock_Hour := #SystemTimeRead.HOUR;
   #CPUClock_Day := #SystemTimeRead.DAY;
   #CPUClock_Month := #SystemTimeRead.MONTH;
   #CPUClock_Year := #SystemTimeRead.YEAR MOD 100; // In the Faceplate we are showing YY format so Moduls the Year(2021 MOD 100 =21) 
   (* ----------------------------------------------------------------- Memory Information -------------------------------------------------------------*)
   (* Memory Card Information *)
   (* Memory Card Information - Memory Available*)

   #GetSMCinfo_Instance(REQ := TRUE,
                        Mode := 0,
                        Done => #dummybool,
                        Busy => #dummybool,
                        Error => #dummybool,
                        Status => #DummyWord,
                        Info := #DummyUDint);
   #DummyDint := UDINT_TO_DINT(#DummyUDint);
   #Memory_Total := #DummyDint * 1024; // (* Step 7 we are getting in Bytes and showing in MB in Faceplate so Multiplied with 1024 *)
   (* Memory Card Information - Memory Used*)
   #GetSMCinfo_Instance_1(REQ := TRUE,
                          Mode := 1,
                          Done => #dummybool,
                          Busy => #dummybool,
                          Error => #dummybool,
                          Status => #DummyWord,
                          Info := #DummyUDint);
   #DummyDint := UDINT_TO_DINT(#DummyUDint);
   IF #GetSMCinfo_Instance_1.Done THEN
       #Memory_Used := #DummyDint * 1024; //(* Step 7 we are getting in Bytes and showing in MB in Faceplate so Multiplied with 1024 *)
   END_IF;
   (* Memory Display in Percentage Display*)
   #DummyReal := DINT_TO_REAL(#Memory_Total);
   #DummyReal1 := DINT_TO_REAL(#Memory_Used);
   IF #DummyReal1 <= #DummyReal THEN
       #Mem_UsePercentage := ((#DummyReal1 / #DummyReal) * 100);
   END_IF;
   (* ----------------------------------------------------------------- CPU Software Information -------------------------------------------------------------*)
   #GET_IM_DATA_Instance(LADDR := 50,
                         IM_TYPE := 0,
                         DONE => #dummybool,
                         BUSY => #dummybool,
                         ERROR => #dummybool,
                         STATUS => #DummyWord,
                         DATA := #DATA);
   (*CPU Software Revision*)
   #Software_RevisionV1 := #DATA.Software_Revision.Functional;
   #Software_RevisionV2 := #DATA.Software_Revision.Bugfix;
   #Software_RevisionV3 := #DATA.Software_Revision.Internal;

   #OUT.CPU_OK := NOT #ALARM_AlarmPresent AND NOT #ALARM_Failure_Ack_Requ;

   IF #CPU_ERROR AND NOT #OUT.Type_Fault AND NOT #ALARM_Failure_Ack_Requ AND (#AlarmNo = 0) THEN
       #StatusWork := 1;
   END_IF;
   (* ----------------------------------------------------------------- Alarm  -------------------------------------------------------------*)
   (*Alarm Present*)
   #ALARM_AlarmPresent := NOT #CPU_ERROR OR #OUT.Type_Fault;
   (*Warning Present*)
   #ALARM_WarnPresent := #AOff;

   (*Skip alarm handling if alarm/warning not present*)
   IF #ALARM_AlarmPresent OR #ALARM_WarnPresent OR #ALARM_Failure_Ack_Requ OR #ALARM_WarnAckRequired OR (#AlarmNo > 0) THEN
       #Clear := #AOn;
       (*Go to Clear Alarm*)
       IF #ALARM_AlarmPresent OR #ALARM_WarnPresent OR #ALARM_Failure_Ack_Requ OR #ALARM_WarnAckRequired OR (#AlarmNo = 0) THEN
           #Ack := #AOff;
           (*Go to Alarm Acknowledge*)
           #dummybool := #ALARM_Failure_Ack_Requ OR #ALARM_WarnAckRequired;
           IF NOT #ALARM_AlarmPresent AND NOT #ALARM_WarnPresent AND #dummybool THEN
               #Ack := #AOn;
           END_IF;
           (*Alarm CPU Type Fault*)
           #dummybool := #OUT.Type_Fault OR (#AlarmNo = 3);
           IF #AlarmNo = 3 OR #OUT.Type_Fault THEN
               #StatusWork := 120;
               #AlarmNo := 3;
               #Ack := #AOn;
           END_IF;
           (*Alarm CPU Error*)
           #dummybool := NOT #CPU_ERROR OR (#AlarmNo = 2);
           IF #AlarmNo = 2 OR NOT #CPU_ERROR THEN
               #StatusWork := 121; // Status Algorithm = 121 (CPU Error), add by asutp 17.11.2024
               #AlarmNo := 2;
               #Ack := #AOn;
           END_IF;
           #Ack := #AOn;
       ELSE
           #Ack := #AOff;
       END_IF;

       (*Alarm Acknowledge*)
       IF #Ack THEN
           IF (#AlarmNo > #AlarmNo_Old) THEN
               IF (#AlarmNo > 1) THEN
                   #ALARM_Failure_Ack_Requ := #AOn;
               ELSE
                   #ALARM_WarnAckRequired := #AOn;
               END_IF;
           END_IF;

           #AlarmNo_Old := #AlarmNo;

           IF #CMD_Acknowledge OR (#AlarmNo = 0) THEN
               #ALARM_Failure_Ack_Requ := #AOff;
               #ALARM_WarnAckRequired := #AOff;
           END_IF;

           IF (#AlarmNo = 0) OR #ALARM_Failure_Ack_Requ OR #ALARM_WarnAckRequired THEN
               #Clear := #AOff;
           END_IF;
       END_IF;
       IF #Clear THEN
           #dummybool := (#AlarmNo = 3) AND NOT #OUT.Type_Fault;
           #dummybool := #dummybool OR ((#AlarmNo = 2) AND #CPU_ERROR);

           IF #dummybool THEN
               #AlarmNo := 0;
           END_IF;

           IF NOT #ALARM_AlarmPresent AND NOT #ALARM_WarnPresent AND NOT #ALARM_Failure_Ack_Requ AND NOT #ALARM_WarnAckRequired AND (#AlarmNo = 0) THEN
               #AlarmNo_Old := 0;
           END_IF;
       END_IF;

   END_IF;

   (* ------------------------------------------------------------------------------------------------------------------------------*)







   (* Bit 16-19: Mode
   0 = Auto
   1= Single Start
   2 = Manual
   3= Local
   4= Test Mode
   *)
   #MSW.EXT.ModeBit1 := 0;
   #MSW.EXT.ModeBit2 := 0;
   #MSW.EXT.ModeBit3 := 0;
   #MSW.EXT.BIT19 := 0;
   #MSW.EXT.BIT20 := 0;
   (*Bit 21 ALARM Suppressed*)
   #MSW.EXT.AlarmSuppressed := 0;


   (*Bit: 22 Alarm Condition Present *)
   #MSW.EXT.AlarmPresent := #ALARM_AlarmPresent;
   (* Bit 23: Alarm Failure Present or Unacknowledged *)
   IF #AlarmNo > 1 OR #ALARM_Failure_Ack_Requ THEN
       #MSW.EXT.AlarmFailUnAck := 1;
   ELSE
       #MSW.EXT.AlarmFailUnAck := 0;
   END_IF;
   (* Bit 24: Alarm Warning Present Or Unacknowledged *)
   #MSW.EXT.AlarmWarnUnAck := 0;
   (*Bit 25: Acknowledge Required *)
   #MSW.EXT.AckRequired := #ALARM_Failure_Ack_Requ;
   (*Bit 26: Maintenence *)
   #MSW.EXT.Maintanence := #CPU_MAINT;
   (*Bit 27: Operation *)
   #MSW.EXT.Operation := #AOff;
   (*Bit 28: Forced *)
   #MSW.EXT.Forced := #AOff;
   (*MSW*)
   #Status_Add := #StatusWork + #StatusBuilder;
   IF #Status_Add <> #MSW_Status_Trans THEN
       #MSW_Status_Trans := #Status_Add;
       #MSW.TimeStamp := #Master_Link.TimeStamp;
   END_IF;
   #MSW.Status := #MSW_Status_Trans;
   (*Move Stat Variables to Out*)
   #CPU_OK := #OUT.CPU_OK;
   #Type_Fault := #OUT.Type_Fault;
END_FUNCTION_BLOCK

FUNCTION_BLOCK "ACESYS_RECIPE"   // FB230, FBD
TITLE = ACESYS V8.0 - Build 002 - RECIPE
{ S7_Optimized_Access := 'FALSE' }
AUTHOR : FLSmidth
FAMILY : ACESYS
NAME : Recipe
VERSION : 8.0
   VAR_INPUT
      CV : Real;   // Setpoint from PID (0.0 - 100.0%)
      F1_QCX : Real;   // QCX Setpoint Feeder 1
      F2_QCX : Real;   // QCX Setpoint Feeder 2
      F3_QCX : Real;   // QCX Setpoint Feeder 3
      F4_QCX : Real;   // QCX Setpoint Feeder 4
      F5_QCX : Real;   // QCX Setpoint Feeder 5
      F6_QCX : Real;   // QCX Setpoint Feeder 6
      F7_QCX : Real;   // QCX Setpoint Feeder 7
      F8_QCX : Real;   // QCX Setpoint Feeder 8
      F1_RUN : Bool;   // Feeder 1 Running
      F2_RUN : Bool;   // Feeder 2 Running
      F3_RUN : Bool;   // Feeder 3 Running
      F4_RUN : Bool;   // Feeder 4 Running
      F5_RUN : Bool;   // Feeder 5 Running
      F6_RUN : Bool;   // Feeder 6 Running
      F7_RUN : Bool;   // Feeder 7 Running
      F8_RUN : Bool;   // Feeder 8 Running
      MILL_ON : Bool;   // Mill and Feeding running
      CCA : Bool;   // Computer Control Accept - permission to use QCX setpoints
   END_VAR
   VAR_OUTPUT
      OK : Bool;   // No fault states
      MAX_OUT : Bool;   // Max. Output reached for at least one feeder
      SPCTL : Bool;   // Setpoint Control (QCX Active)
      CV_ENG : Real;   // Total Feed Set Point (t/h)
      F1_ENG : Real;   // Setpoint Feeder 1 (t/h)
      F2_ENG : Real;   // Setpoint Feeder 2 (t/h)
      F3_ENG : Real;   // Setpoint Feeder 3 (t/h)
      F4_ENG : Real;   // Setpoint Feeder 4 (t/h)
      F5_ENG : Real;   // Setpoint Feeder 5 (t/h)
      F6_ENG : Real;   // Setpoint Feeder 6 (t/h)
      F7_ENG : Real;   // Setpoint Feeder 7 (t/h)
      F8_ENG : Real;   // Setpoint Feeder 8 (t/h)
      F1_PCT : Real;   // Setpoint Feeder 1 (%)
      F2_PCT : Real;   // Setpoint Feeder 2 (%)
      F3_PCT : Real;   // Setpoint Feeder 3 (%)
      F4_PCT : Real;   // Setpoint Feeder 4 (%)
      F5_PCT : Real;   // Setpoint Feeder 5 (%)
      F6_PCT : Real;   // Setpoint Feeder 6 (%)
      F7_PCT : Real;   // Setpoint Feeder 7 (%)
      F8_PCT : Real;   // Setpoint Feeder 8 (%)
      MSW : "ACESYS_HMI_STAT_32T";
   END_VAR
   VAR_IN_OUT
      KA : Bool;   // Keep Alive - Communication Watchdog
      SEL : Bool;   // Select QCX
      TOKEN : "ACESYS_TOKEN";
   END_VAR
   VAR
      BlockInfo : Struct
         Ace_Version : Int;   // Acesys Block Version Number
         Ace_BuildNo : Int;   // Acesys Block Build Number
         DB_Number : Int;   // Block Instance DB Number
      END_STRUCT;
      FP_CMD : Struct   // Faceplate Commands
         Spare_08 : Bool;
         Spare_09 : Bool;
         Spare_10 : Bool;
         Spare_11 : Bool;
         Spare_12 : Bool;
         Spare_13 : Bool;
         Spare_14 : Bool;
         AckAlarm : Bool;   // Alarm Acknowledge
         Spare_00 : Bool;
         Spare_01 : Bool;
         Spare_02 : Bool;
         Spare_03 : Bool;
         Spare_04 : Bool;
         Spare_05 : Bool;
         Spare_06 : Bool;
         Spare_07 : Bool;
      END_STRUCT;
      FP_SEL : Struct
         Rcp01 : Bool;
         Rcp02 : Bool;
         Rcp03 : Bool;
         Rcp04 : Bool;
         Rcp05 : Bool;
         Rcp06 : Bool;
         Rcp07 : Bool;
         Rcp08 : Bool;
         Accept_Rcp : Bool;   // Accept Selected Recipe
      END_STRUCT;
      FP_EN : Struct
         Force_Feeder1 : Bool;   // Force Feeder 1 from faceplate
         Force_Feeder2 : Bool;   // Force Feeder 2 from faceplate
         Force_Feeder3 : Bool;   // Force Feeder 3 from faceplate
         Force_Feeder4 : Bool;   // Force Feeder 4 from faceplate
         Force_Feeder5 : Bool;   // Force Feeder 5 from faceplate
         Force_Feeder6 : Bool;   // Force Feeder 6 from faceplate
         Force_Feeder7 : Bool;   // Force Feeder 7 from faceplate
         Force_Feeder8 : Bool;   // Force Feeder 8 from faceplate
         KA : Bool;   // Enable Keep Alive Supervison
         QCX : Bool;   // Enable QCX
      END_STRUCT;
      FP_RARM : Struct
         Force_Values : Array[1..8] of Real;   // Force values from ECS (t/h)
         Recipe : Array[1..7, 2..8] of Real;   // Recipe area: Recipe 1..8 - feeder 2..8 (Feeder 1 calculated)
         Recipe_Selected : Array[1..8] of Real;   // Selected Recipe: Feeder 1..8
         Recipe_Accepted : Array[1..8] of Real;   // Accepted Recipe: Feeder 1..8
         Q_T : Real := 500.0;   // Max Setpoint total feed (t/h)
         Q_F1 : Real := 250.0;   // Feeder 1 total feed (t/h), clinker
         Q_F2 : Real := 50.0;   // Feeder 2 total feed (t/h)
         Q_F3 : Real;   // Feeder 3 total feed (t/h)
         Q_F4 : Real;   // Feeder 4 total feed (t/h)
         Q_F5 : Real;   // Feeder 5 total feed (t/h)
         Q_F6 : Real;   // Feeder 6 total feed (t/h)
         Q_F7 : Real;   // Feeder 7 total feed (t/h)
         Q_F8 : Real;   // Feeder 8 total feed (t/h)
         QCX_MaxTolerance : Real := 1.0;   // Max. tolerance sum QCX SP / 100%
         KA_Time_PRE : Int := 60;
         KA_Time_ACC : Int;
         NoOfFeeders : Int;   // Number of Feeders
         Max_Output_Feeder1 : Bool;   // Max. output reached feeder 1
         Max_Output_Feeder2 : Bool;   // Max. output reached feeder 2
         Max_Output_Feeder3 : Bool;   // Max. output reached feeder 3
         Max_Output_Feeder4 : Bool;   // Max. output reached feeder 4
         Max_Output_Feeder5 : Bool;   // Max. output reached feeder 5
         Max_Output_Feeder6 : Bool;   // Max. output reached feeder 6
         Max_Output_Feeder7 : Bool;   // Max. output reached feeder 7
         Max_Output_Feeder8 : Bool;   // Max. output reached feeder 8
      END_STRUCT;
      ONS : Struct
         SelOn : Bool;
         SelOff : Bool;
      END_STRUCT;
      KA_Time_MEM : Int;   // Actual Watchdog time left
      FP_SelAcpRcp : Int;
      PB_Time_MEM : Int;
      SelectedRecipeNo : Int;
      TimeQCXsum_MEM : Int;
      StatusWork : Int;   // MSW to ECS
      Sel_Rcp01_Done : Bool;   // Recipe 01 Selected Done
      Sel_Rcp02_Done : Bool;   // Recipe 02 Selected Done
      Sel_Rcp03_Done : Bool;   // Recipe 03 Selected Done
      Sel_Rcp04_Done : Bool;   // Recipe 04 Selected Done
      Sel_Rcp05_Done : Bool;   // Recipe 05 Selected Done
      Sel_Rcp06_Done : Bool;   // Recipe 06 Selected Done
      Sel_Rcp07_Done : Bool;   // Recipe 07 Selected Done
      Accept_Rcp_Done : Bool;   // Accept Selected Recipe Done
      Error_Sum_Ratio_QCX : Bool;
      CMD_AckAlarm : Bool;
      Trig_QCX_CCA : Bool;
      Trig_QCX_KA : Bool;
      Trig_Sum_Ratio : Bool;
      Trig_Sum_Ratio_QCX : Bool;
      Trig_MaxOut : Bool;
      ALARM_AlarmPresent : Bool;
      ALARM_FailureAckRequired : Bool;
      AlarmNo : Int;
      AlarmNo_Old : Int;
      OUT : Struct
         OK : Bool;
         MAX_OUT : Bool;
         SPCTL : Bool;
         CV_ENG : Real;
         F1_ENG : Real;
         F2_ENG : Real;
         F3_ENG : Real;
         F4_ENG : Real;
         F5_ENG : Real;
         F6_ENG : Real;
         F7_ENG : Real;
         F8_ENG : Real;
         F1_PCT : Real;
         F2_PCT : Real;
         F3_PCT : Real;
         F4_PCT : Real;
         F5_PCT : Real;
         F6_PCT : Real;
         F7_PCT : Real;
         F8_PCT : Real;
      END_STRUCT;
      MSW_Status_Trans : Int;
   END_VAR
   VAR_TEMP
      Aon : Bool;
      Aoff : Bool;
      Sum_Feeder : Real;
      Diff_QCX_100 : Real;
      KeepAliveTimeDone : Bool;
      Reset_Select_PB : Bool;
      DummyBool : Bool;
      DummyInt : Int;
   END_VAR
   VAR_TEMP   // added for the SCL form of the ladder/FBD networks
      _w1 : Bool;
      _w2 : Bool;
      _w3 : Bool;
      _w4 : Bool;
      _w5 : Bool;
      _w6 : Bool;
      _w7 : Bool;
      _w8 : Bool;
   END_VAR
BEGIN

REGION Network 1: Always On
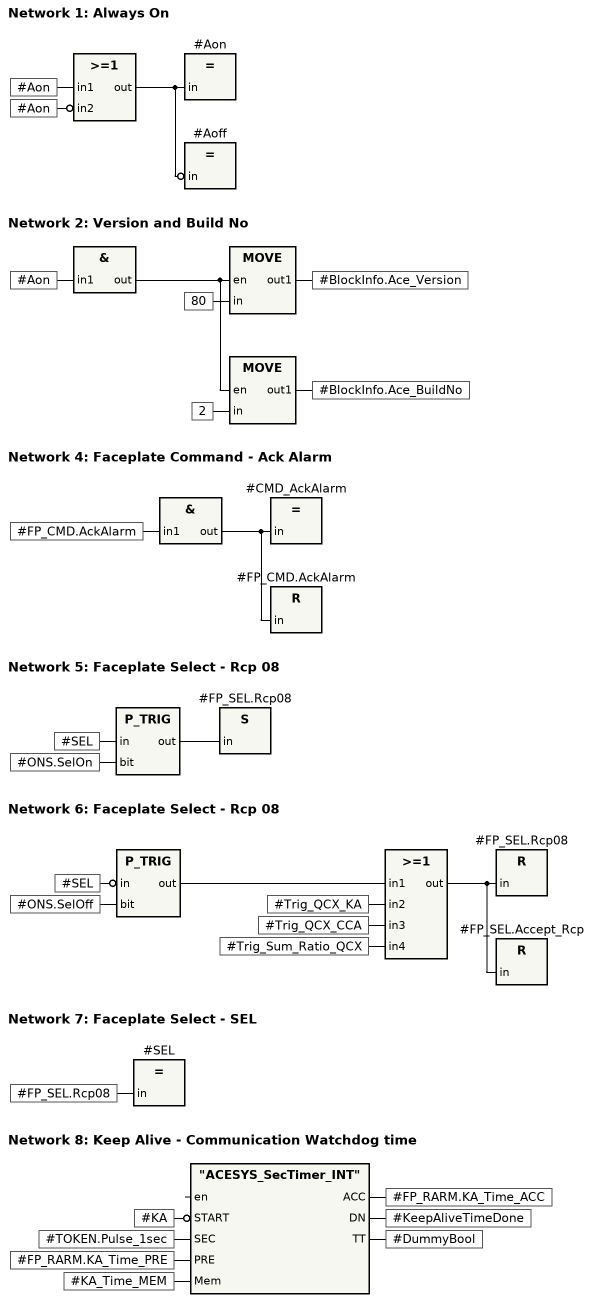
   #Aon := #Aon OR NOT #Aon;
   #Aoff := NOT #Aon;
END_REGION

REGION Network 2: Version and Build No
   IF #Aon THEN
       #BlockInfo.Ace_Version := 80;
       #BlockInfo.Ace_BuildNo := 2;
   END_IF;
END_REGION

REGION Network 3 (STL): Instance DB Number to Faceplate
         L     DINO;
         T     #BlockInfo.DB_Number;
END_REGION

REGION Network 4: Faceplate Command - Ack Alarm
   #CMD_AckAlarm := #FP_CMD.AckAlarm;
   IF #FP_CMD.AckAlarm THEN #FP_CMD.AckAlarm := FALSE; END_IF;
END_REGION

REGION Network 5: Faceplate Select - Rcp 08
   #_w1 := #SEL AND NOT #ONS.SelOn;   // rising edge
   #ONS.SelOn := #SEL;
   IF #_w1 THEN #FP_SEL.Rcp08 := TRUE; END_IF;
END_REGION

REGION Network 6: Faceplate Select - Rcp 08
   #_w1 := NOT #SEL AND NOT #ONS.SelOff;   // rising edge
   #ONS.SelOff := NOT #SEL;
   IF #_w1 OR #Trig_QCX_KA OR #Trig_QCX_CCA OR #Trig_Sum_Ratio_QCX THEN
       #FP_SEL.Rcp08 := FALSE;
       #FP_SEL.Accept_Rcp := FALSE;
   END_IF;
END_REGION

REGION Network 7: Faceplate Select - SEL
   #SEL := #FP_SEL.Rcp08;
END_REGION

REGION Network 8: Keep Alive - Communication Watchdog time
   "ACESYS_SecTimer_INT"(START := NOT #KA,
                         SEC := #TOKEN.Pulse_1sec,
                         PRE := #FP_RARM.KA_Time_PRE,
                         Mem := #KA_Time_MEM,
                         ACC => #FP_RARM.KA_Time_ACC,
                         DN => #KeepAliveTimeDone,
                         TT => #DummyBool);
END_REGION

REGION Network 9: Reset KA-signal after reset of timer
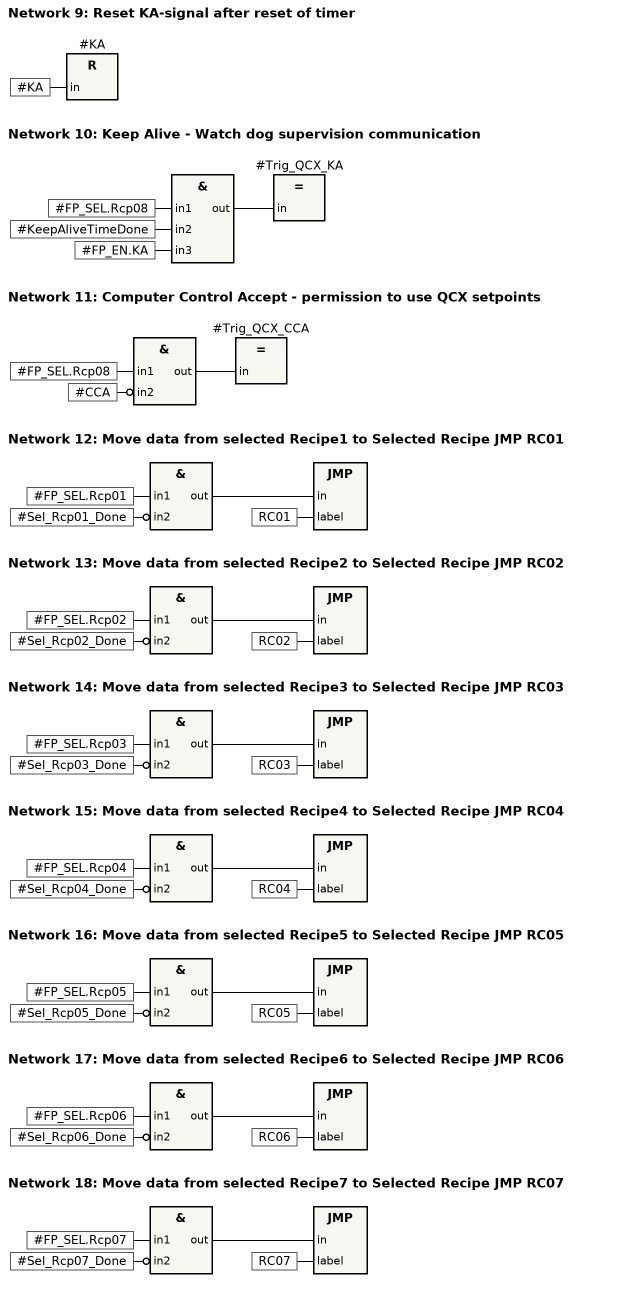
   IF #KA THEN #KA := FALSE; END_IF;
END_REGION

REGION Network 10: Keep Alive - Watch dog supervision communication
   #Trig_QCX_KA := #FP_SEL.Rcp08 AND #KeepAliveTimeDone AND #FP_EN.KA;
END_REGION

REGION Network 11: Computer Control Accept - permission to use QCX setpoints
   #Trig_QCX_CCA := #FP_SEL.Rcp08 AND NOT #CCA;
END_REGION

REGION Network 12: Move data from selected Recipe1 to Selected Recipe JMP RC01
   IF #FP_SEL.Rcp01 AND NOT #Sel_Rcp01_Done THEN GOTO RC01; END_IF;
END_REGION

REGION Network 13: Move data from selected Recipe2 to Selected Recipe JMP RC02
   IF #FP_SEL.Rcp02 AND NOT #Sel_Rcp02_Done THEN GOTO RC02; END_IF;
END_REGION

REGION Network 14: Move data from selected Recipe3 to Selected Recipe JMP RC03
   IF #FP_SEL.Rcp03 AND NOT #Sel_Rcp03_Done THEN GOTO RC03; END_IF;
END_REGION

REGION Network 15: Move data from selected Recipe4 to Selected Recipe JMP RC04
   IF #FP_SEL.Rcp04 AND NOT #Sel_Rcp04_Done THEN GOTO RC04; END_IF;
END_REGION

REGION Network 16: Move data from selected Recipe5 to Selected Recipe JMP RC05
   IF #FP_SEL.Rcp05 AND NOT #Sel_Rcp05_Done THEN GOTO RC05; END_IF;
END_REGION

REGION Network 17: Move data from selected Recipe6 to Selected Recipe JMP RC06
   IF #FP_SEL.Rcp06 AND NOT #Sel_Rcp06_Done THEN GOTO RC06; END_IF;
END_REGION

REGION Network 18: Move data from selected Recipe7 to Selected Recipe JMP RC07
   IF #FP_SEL.Rcp07 AND NOT #Sel_Rcp07_Done THEN GOTO RC07; END_IF;
END_REGION

REGION Network 19: Move data from selected Recipe8 to Selected Recipe JMP RC08
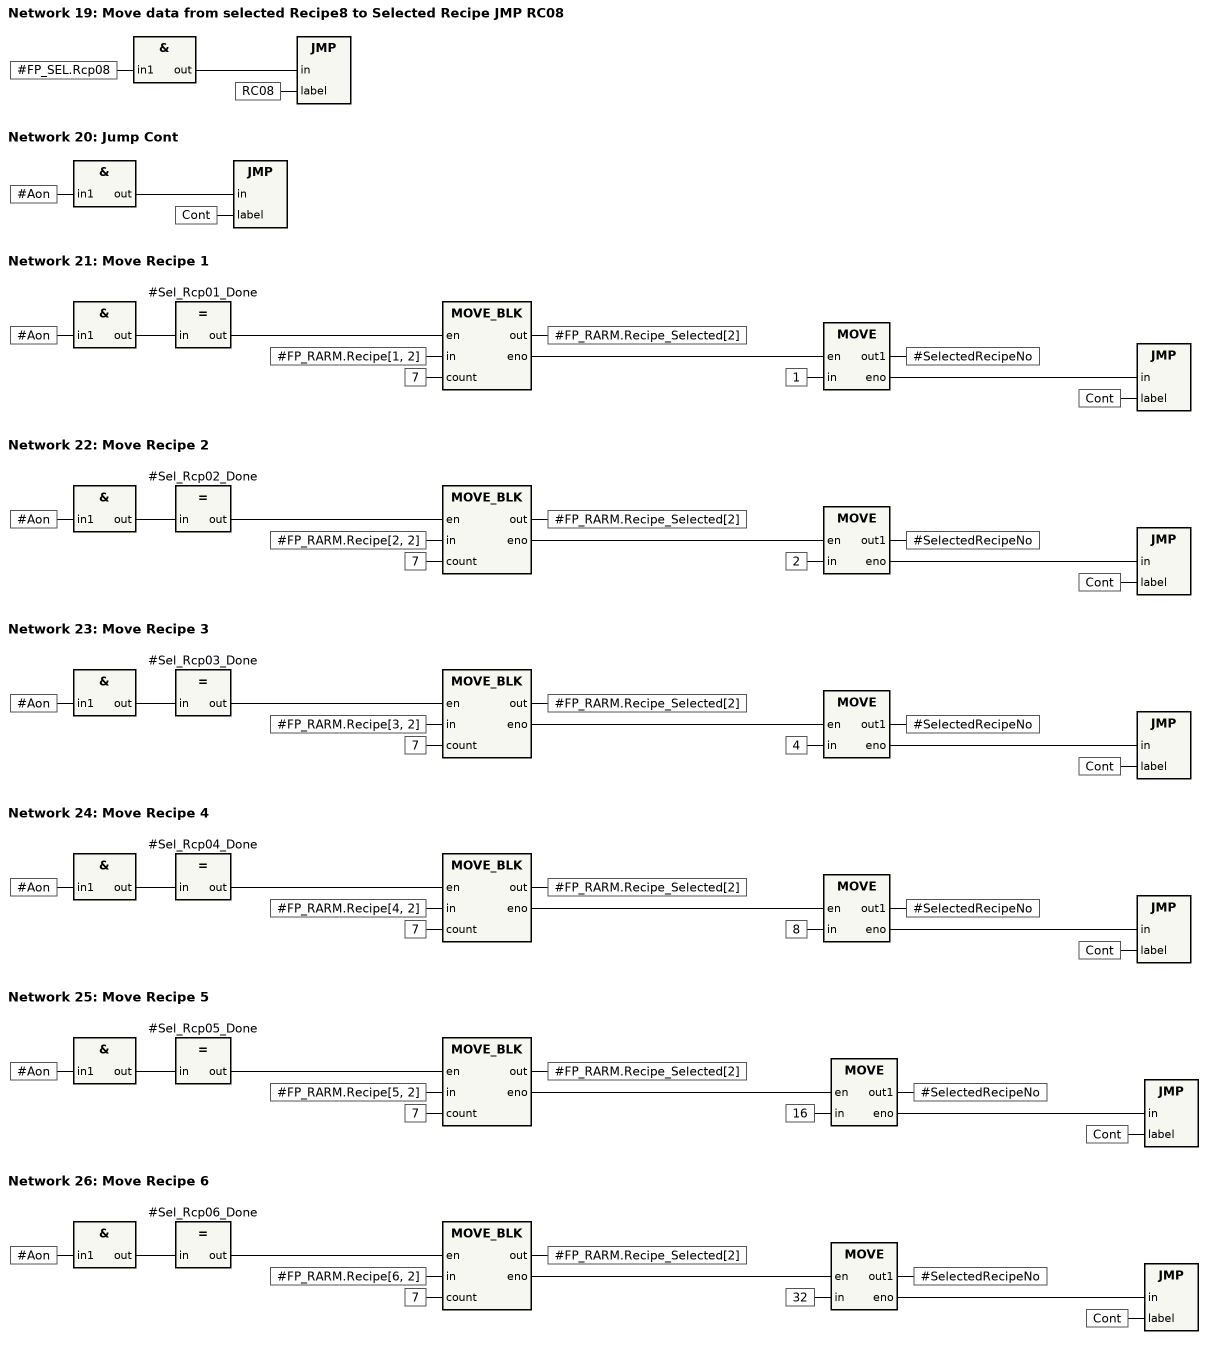
   IF #FP_SEL.Rcp08 THEN GOTO RC08; END_IF;
END_REGION

REGION Network 20: Jump Cont
   IF #Aon THEN GOTO Cont; END_IF;
END_REGION

REGION Network 21: Move Recipe 1
   // Build 002 - 24 Jun 2019 (EXTBOB) : Selected Receipe Number moved to #SelectedRecipeNo variable
   RC01:
   #Sel_Rcp01_Done := #Aon;
   IF #Aon THEN
       MOVE_BLK(IN := #FP_RARM.Recipe[1, 2], COUNT := 7, OUT => #FP_RARM.Recipe_Selected[2]);
       #SelectedRecipeNo := 1;
       GOTO Cont;
   END_IF;
END_REGION

REGION Network 22: Move Recipe 2
   // Build 002 - 24 Jun 2019 (EXTBOB) : Selected Receipe Number moved to #SelectedRecipeNo variable
   RC02:
   #Sel_Rcp02_Done := #Aon;
   IF #Aon THEN
       MOVE_BLK(IN := #FP_RARM.Recipe[2, 2], COUNT := 7, OUT => #FP_RARM.Recipe_Selected[2]);
       #SelectedRecipeNo := 2;
       GOTO Cont;
   END_IF;
END_REGION

REGION Network 23: Move Recipe 3
   // Build 002 - 24 Jun 2019 (EXTBOB) : Selected Receipe Number moved to #SelectedRecipeNo variable
   RC03:
   #Sel_Rcp03_Done := #Aon;
   IF #Aon THEN
       MOVE_BLK(IN := #FP_RARM.Recipe[3, 2], COUNT := 7, OUT => #FP_RARM.Recipe_Selected[2]);
       #SelectedRecipeNo := 4;
       GOTO Cont;
   END_IF;
END_REGION

REGION Network 24: Move Recipe 4
   // Build 002 - 24 Jun 2019 (EXTBOB) : Selected Receipe Number moved to #SelectedRecipeNo variable
   RC04:
   #Sel_Rcp04_Done := #Aon;
   IF #Aon THEN
       MOVE_BLK(IN := #FP_RARM.Recipe[4, 2], COUNT := 7, OUT => #FP_RARM.Recipe_Selected[2]);
       #SelectedRecipeNo := 8;
       GOTO Cont;
   END_IF;
END_REGION

REGION Network 25: Move Recipe 5
   // Build 002 - 24 Jun 2019 (EXTBOB) : Selected Receipe Number moved to #SelectedRecipeNo variable
   RC05:
   #Sel_Rcp05_Done := #Aon;
   IF #Aon THEN
       MOVE_BLK(IN := #FP_RARM.Recipe[5, 2], COUNT := 7, OUT => #FP_RARM.Recipe_Selected[2]);
       #SelectedRecipeNo := 16;
       GOTO Cont;
   END_IF;
END_REGION

REGION Network 26: Move Recipe 6
   // Build 002 - 24 Jun 2019 (EXTBOB) : Selected Receipe Number moved to #SelectedRecipeNo variable
   RC06:
   #Sel_Rcp06_Done := #Aon;
   IF #Aon THEN
       MOVE_BLK(IN := #FP_RARM.Recipe[6, 2], COUNT := 7, OUT => #FP_RARM.Recipe_Selected[2]);
       #SelectedRecipeNo := 32;
       GOTO Cont;
   END_IF;
END_REGION

REGION Network 27: Move Recipe 7
   // Build 002 - 24 Jun 2019 (EXTBOB) : Selected Receipe Number moved to #SelectedRecipeNo variable
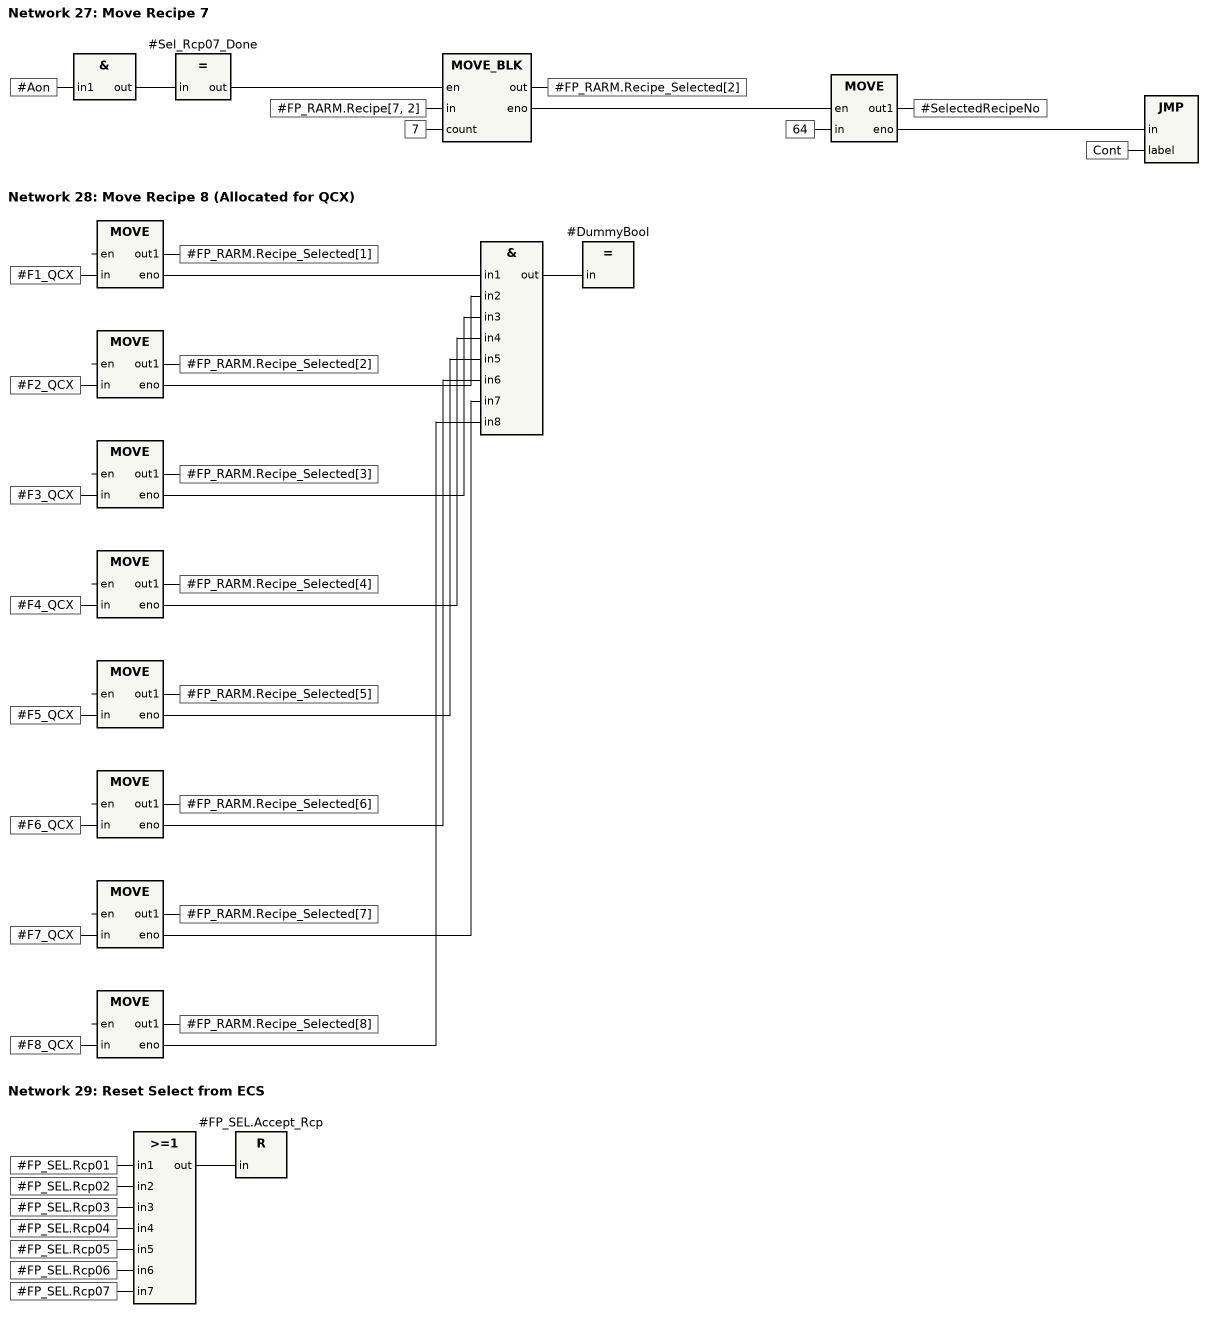
   RC07:
   #Sel_Rcp07_Done := #Aon;
   IF #Aon THEN
       MOVE_BLK(IN := #FP_RARM.Recipe[7, 2], COUNT := 7, OUT => #FP_RARM.Recipe_Selected[2]);
       #SelectedRecipeNo := 64;
       GOTO Cont;
   END_IF;
END_REGION

REGION Network 28: Move Recipe 8 (Allocated for QCX)
   RC08:
   #FP_RARM.Recipe_Selected[1] := #F1_QCX;
   #FP_RARM.Recipe_Selected[2] := #F2_QCX;
   #FP_RARM.Recipe_Selected[3] := #F3_QCX;
   #FP_RARM.Recipe_Selected[4] := #F4_QCX;
   #FP_RARM.Recipe_Selected[5] := #F5_QCX;
   #FP_RARM.Recipe_Selected[6] := #F6_QCX;
   #FP_RARM.Recipe_Selected[7] := #F7_QCX;
   #FP_RARM.Recipe_Selected[8] := #F8_QCX;
   #DummyBool := TRUE;
END_REGION

REGION Network 29: Reset Select from ECS
   Cont:
   IF #FP_SEL.Rcp01 OR #FP_SEL.Rcp02 OR #FP_SEL.Rcp03 OR #FP_SEL.Rcp04 OR #FP_SEL.Rcp05 OR #FP_SEL.Rcp06 OR #FP_SEL.Rcp07 THEN
       #FP_SEL.Accept_Rcp := FALSE;
   END_IF;
END_REGION

REGION Network 30: Reset Select PB Timer
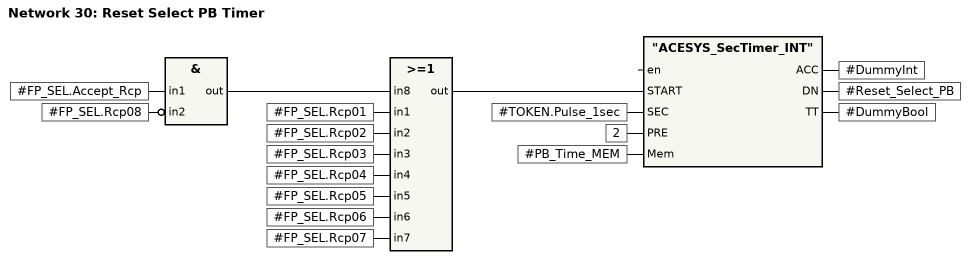
   "ACESYS_SecTimer_INT"(START := (#FP_SEL.Accept_Rcp AND NOT #FP_SEL.Rcp08) OR #FP_SEL.Rcp01 OR #FP_SEL.Rcp02 OR #FP_SEL.Rcp03 OR #FP_SEL.Rcp04 OR #FP_SEL.Rcp05 OR #FP_SEL.Rcp06 OR #FP_SEL.Rcp07,
                         SEC := #TOKEN.Pulse_1sec,
                         PRE := 2,
                         Mem := #PB_Time_MEM,
                         ACC => #DummyInt,
                         DN => #Reset_Select_PB,
                         TT => #DummyBool);
END_REGION

REGION Network 31: Reset Select Recipe
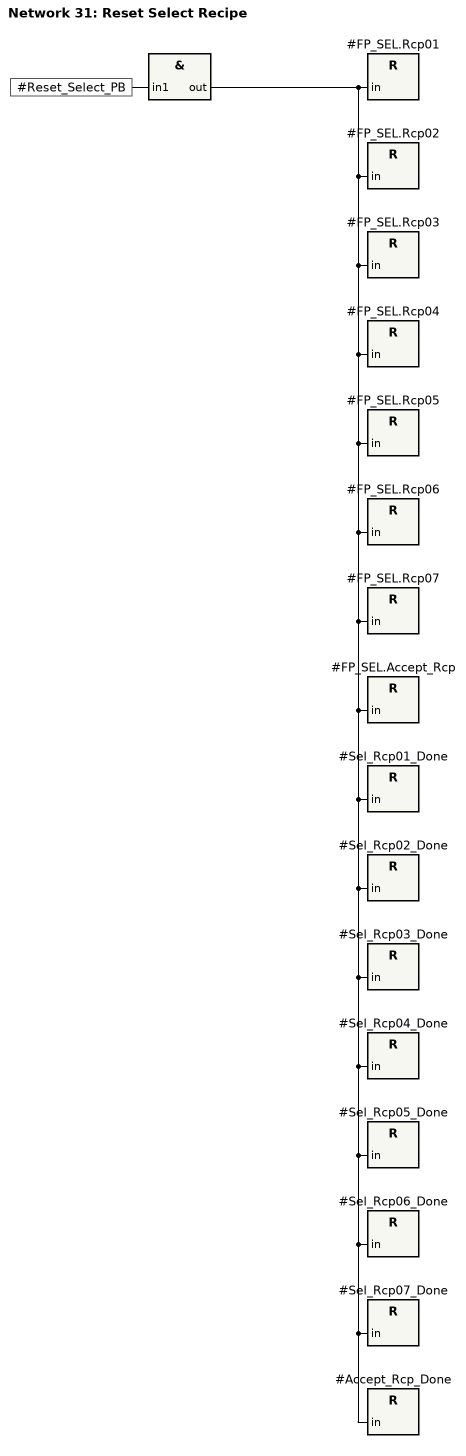
   IF #Reset_Select_PB THEN
       #FP_SEL.Rcp01 := FALSE;
       #FP_SEL.Rcp02 := FALSE;
       #FP_SEL.Rcp03 := FALSE;
       #FP_SEL.Rcp04 := FALSE;
       #FP_SEL.Rcp05 := FALSE;
       #FP_SEL.Rcp06 := FALSE;
       #FP_SEL.Rcp07 := FALSE;
       #FP_SEL.Accept_Rcp := FALSE;
       #Sel_Rcp01_Done := FALSE;
       #Sel_Rcp02_Done := FALSE;
       #Sel_Rcp03_Done := FALSE;
       #Sel_Rcp04_Done := FALSE;
       #Sel_Rcp05_Done := FALSE;
       #Sel_Rcp06_Done := FALSE;
       #Sel_Rcp07_Done := FALSE;
       #Accept_Rcp_Done := FALSE;
   END_IF;
END_REGION

REGION Network 32: Calculate Setp. Feeder 1
   // Calculate only feeder 1 if QCX not selected
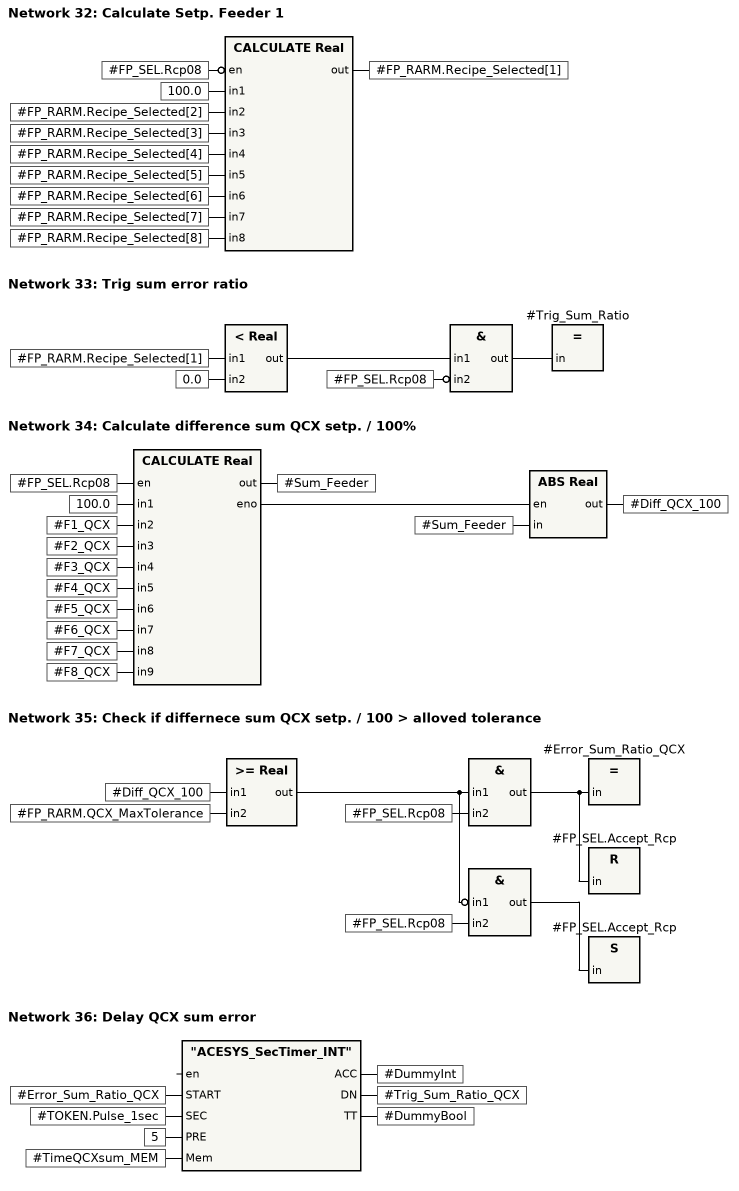
   IF NOT #FP_SEL.Rcp08 THEN
       #FP_RARM.Recipe_Selected[1] := 100.0-(#FP_RARM.Recipe_Selected[2]+#FP_RARM.Recipe_Selected[3]+#FP_RARM.Recipe_Selected[4]+#FP_RARM.Recipe_Selected[5]+#FP_RARM.Recipe_Selected[6]+#FP_RARM.Recipe_Selected[7]+#FP_RARM.Recipe_Selected[8]);
   END_IF;
END_REGION

REGION Network 33: Trig sum error ratio
   #Trig_Sum_Ratio := (#FP_RARM.Recipe_Selected[1] < 0.0) AND NOT #FP_SEL.Rcp08;
END_REGION

REGION Network 34: Calculate difference sum QCX setp. / 100%
   IF #FP_SEL.Rcp08 THEN
       #Sum_Feeder := 100.0-(#F1_QCX+#F2_QCX+#F3_QCX+#F4_QCX+#F5_QCX+#F6_QCX+#F7_QCX+#F8_QCX);
       #Diff_QCX_100 := ABS(#Sum_Feeder);
   END_IF;
END_REGION

REGION Network 35: Check if differnece sum QCX setp. / 100 > alloved tolerance
   #_w1 := #Diff_QCX_100 >= #FP_RARM.QCX_MaxTolerance;
   #Error_Sum_Ratio_QCX := #_w1 AND #FP_SEL.Rcp08;
   IF #Error_Sum_Ratio_QCX THEN #FP_SEL.Accept_Rcp := FALSE; END_IF;
   IF NOT #_w1 AND #FP_SEL.Rcp08 THEN #FP_SEL.Accept_Rcp := TRUE; END_IF;
END_REGION

REGION Network 36: Delay QCX sum error
   "ACESYS_SecTimer_INT"(START := #Error_Sum_Ratio_QCX,
                         SEC := #TOKEN.Pulse_1sec,
                         PRE := 5,
                         Mem := #TimeQCXsum_MEM,
                         ACC => #DummyInt,
                         DN => #Trig_Sum_Ratio_QCX,
                         TT => #DummyBool);
END_REGION

REGION Network 37: Accept Recipe
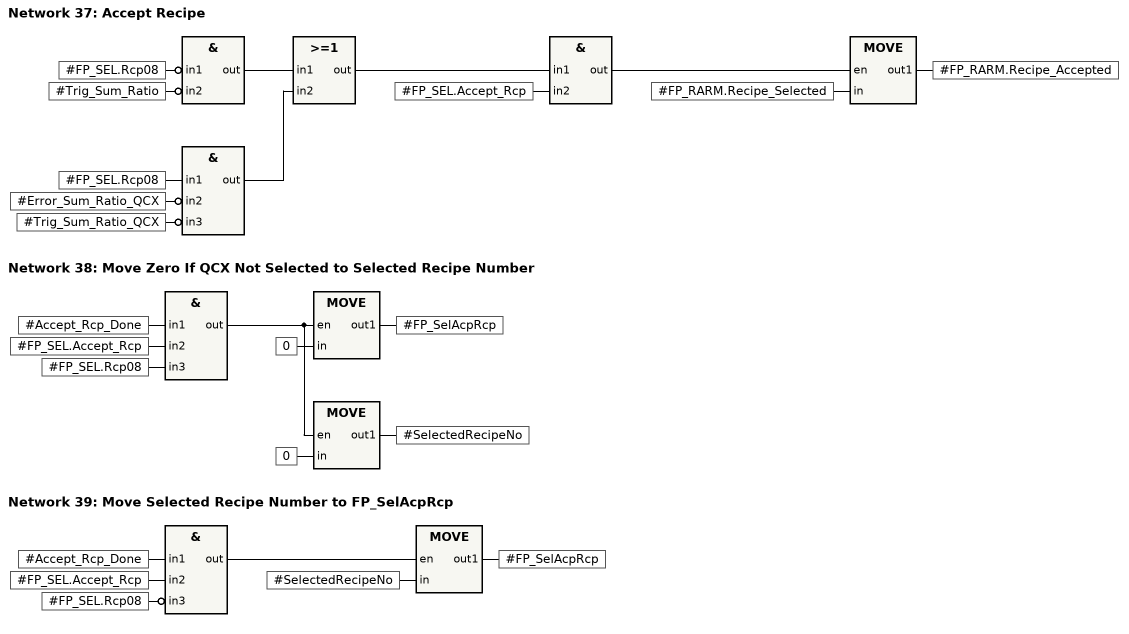
   IF ((NOT #FP_SEL.Rcp08 AND NOT #Trig_Sum_Ratio) OR (#FP_SEL.Rcp08 AND NOT #Error_Sum_Ratio_QCX AND NOT #Trig_Sum_Ratio_QCX)) AND #FP_SEL.Accept_Rcp THEN
       #FP_RARM.Recipe_Accepted := #FP_RARM.Recipe_Selected;
   END_IF;
END_REGION

REGION Network 38: Move Zero If QCX Not Selected to Selected Recipe Number
   // Build 002 - 24 Jun 2019 (EXTBOB) : If QCX selected then Zero moved to Selected Receipe Number & #FP_SelAcpRcp variable
   IF #Accept_Rcp_Done AND #FP_SEL.Accept_Rcp AND #FP_SEL.Rcp08 THEN
       #FP_SelAcpRcp := 0;
       #SelectedRecipeNo := 0;
   END_IF;
END_REGION

REGION Network 39: Move Selected Recipe Number to FP_SelAcpRcp
   // Build 002 - 24 Jun 2019 (EXTBOB) : Selected Receipe Number moved to #FP_SelAcpRcp variable for ECS selectedAccepted recipe display
   IF #Accept_Rcp_Done AND #FP_SEL.Accept_Rcp AND NOT #FP_SEL.Rcp08 THEN
       #FP_SelAcpRcp := #SelectedRecipeNo;
   END_IF;
END_REGION

REGION Network 40: Clamp Force Values to feeder max
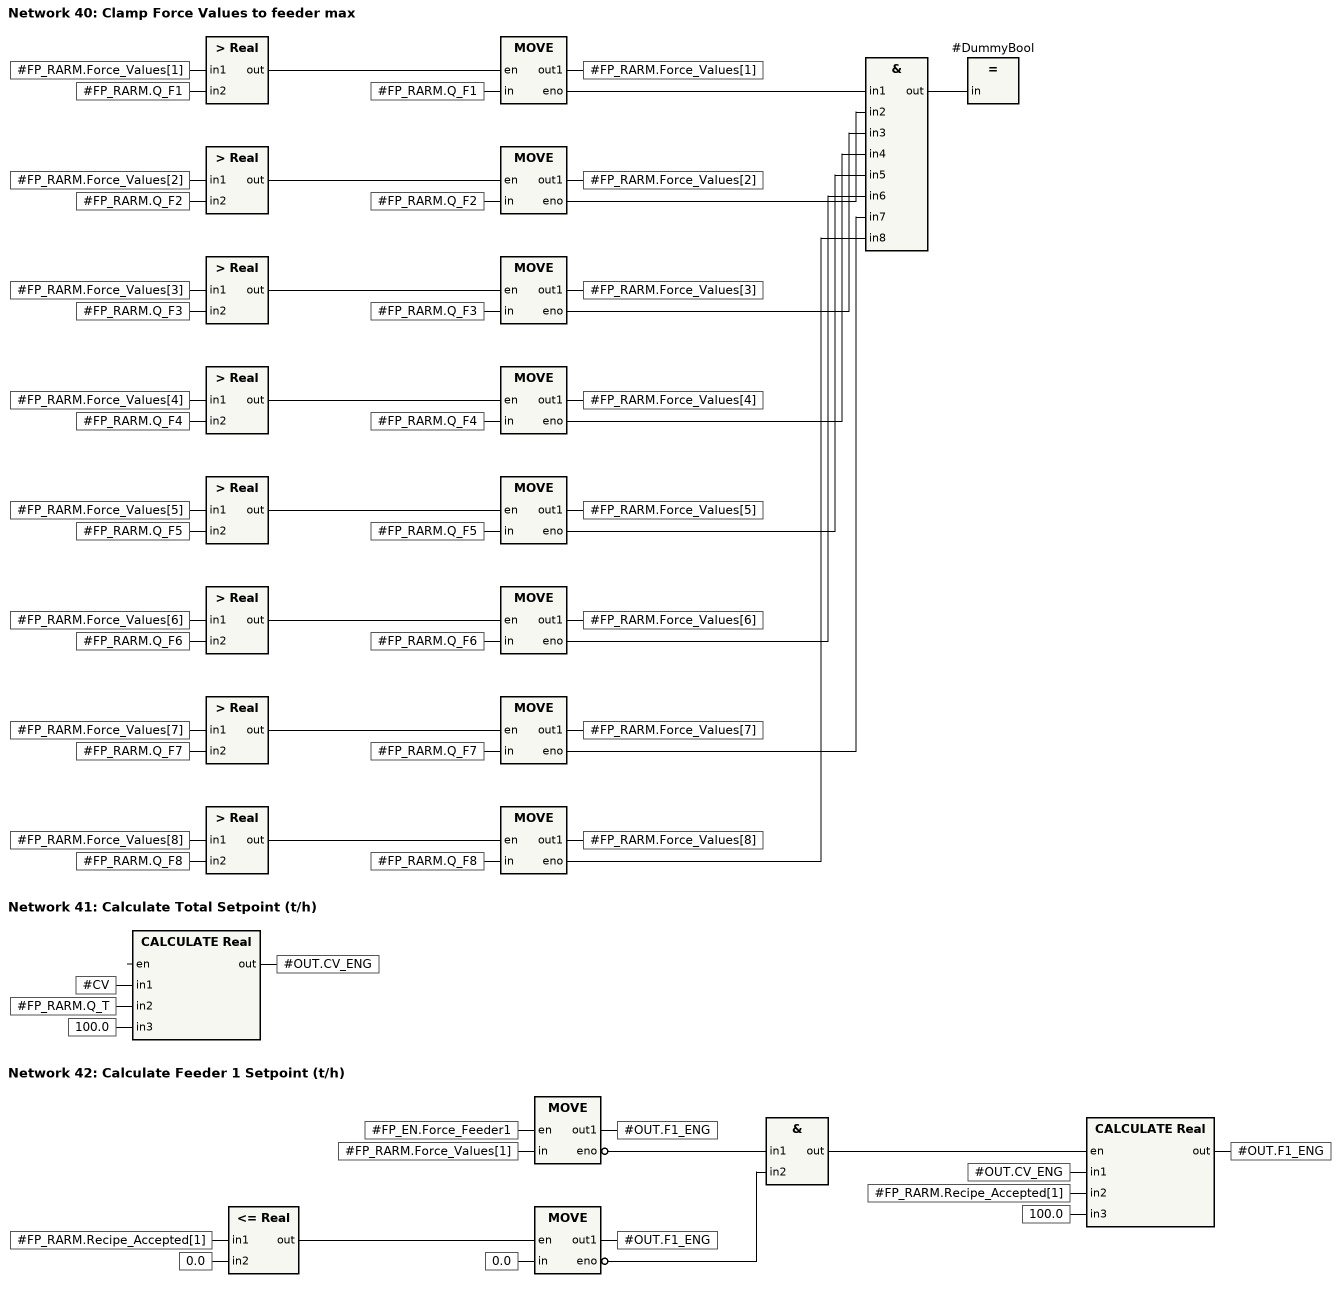
   // ENO of a box is taken as its EN; it also drops when the box reports an error
   #_w1 := #FP_RARM.Force_Values[1] > #FP_RARM.Q_F1;
   IF #_w1 THEN #FP_RARM.Force_Values[1] := #FP_RARM.Q_F1; END_IF;
   #_w2 := #FP_RARM.Force_Values[2] > #FP_RARM.Q_F2;
   IF #_w2 THEN #FP_RARM.Force_Values[2] := #FP_RARM.Q_F2; END_IF;
   #_w3 := #FP_RARM.Force_Values[3] > #FP_RARM.Q_F3;
   IF #_w3 THEN #FP_RARM.Force_Values[3] := #FP_RARM.Q_F3; END_IF;
   #_w4 := #FP_RARM.Force_Values[4] > #FP_RARM.Q_F4;
   IF #_w4 THEN #FP_RARM.Force_Values[4] := #FP_RARM.Q_F4; END_IF;
   #_w5 := #FP_RARM.Force_Values[5] > #FP_RARM.Q_F5;
   IF #_w5 THEN #FP_RARM.Force_Values[5] := #FP_RARM.Q_F5; END_IF;
   #_w6 := #FP_RARM.Force_Values[6] > #FP_RARM.Q_F6;
   IF #_w6 THEN #FP_RARM.Force_Values[6] := #FP_RARM.Q_F6; END_IF;
   #_w7 := #FP_RARM.Force_Values[7] > #FP_RARM.Q_F7;
   IF #_w7 THEN #FP_RARM.Force_Values[7] := #FP_RARM.Q_F7; END_IF;
   #_w8 := #FP_RARM.Force_Values[8] > #FP_RARM.Q_F8;
   IF #_w8 THEN #FP_RARM.Force_Values[8] := #FP_RARM.Q_F8; END_IF;
   #DummyBool := #_w1 AND #_w2 AND #_w3 AND #_w4 AND #_w5 AND #_w6 AND #_w7 AND #_w8;
END_REGION

REGION Network 41: Calculate Total Setpoint (t/h)
   #OUT.CV_ENG := (#CV*#FP_RARM.Q_T)/100.0;
END_REGION

REGION Network 42: Calculate Feeder 1 Setpoint (t/h)
   IF #FP_EN.Force_Feeder1 THEN #OUT.F1_ENG := #FP_RARM.Force_Values[1]; END_IF;
   #_w1 := #FP_RARM.Recipe_Accepted[1] <= 0.0;
   IF #_w1 THEN #OUT.F1_ENG := 0.0; END_IF;
   IF NOT #FP_EN.Force_Feeder1 AND NOT #_w1 THEN
       #OUT.F1_ENG := (#OUT.CV_ENG*#FP_RARM.Recipe_Accepted[1])/100.0;
   END_IF;
END_REGION

REGION Network 43: Calculate Feeder 2 Setpoint (t/h)
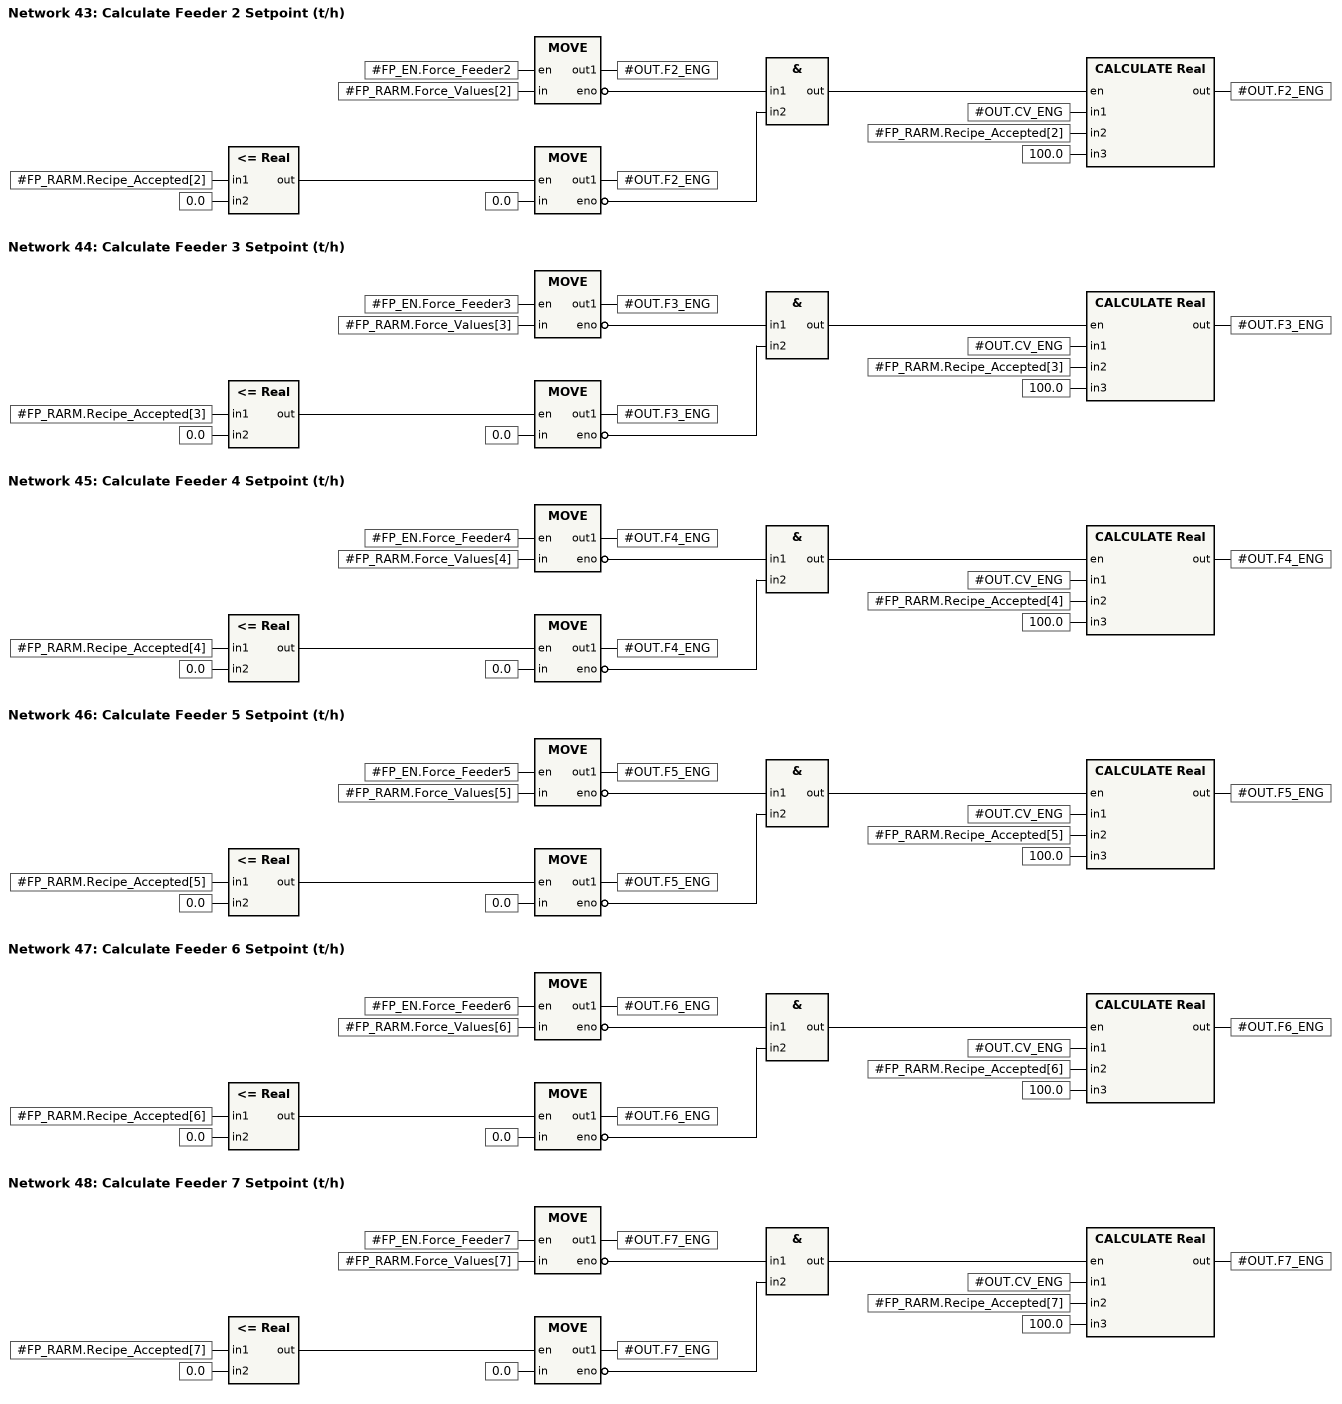
   IF #FP_EN.Force_Feeder2 THEN #OUT.F2_ENG := #FP_RARM.Force_Values[2]; END_IF;
   #_w1 := #FP_RARM.Recipe_Accepted[2] <= 0.0;
   IF #_w1 THEN #OUT.F2_ENG := 0.0; END_IF;
   IF NOT #FP_EN.Force_Feeder2 AND NOT #_w1 THEN
       #OUT.F2_ENG := (#OUT.CV_ENG*#FP_RARM.Recipe_Accepted[2])/100.0;
   END_IF;
END_REGION

REGION Network 44: Calculate Feeder 3 Setpoint (t/h)
   IF #FP_EN.Force_Feeder3 THEN #OUT.F3_ENG := #FP_RARM.Force_Values[3]; END_IF;
   #_w1 := #FP_RARM.Recipe_Accepted[3] <= 0.0;
   IF #_w1 THEN #OUT.F3_ENG := 0.0; END_IF;
   IF NOT #FP_EN.Force_Feeder3 AND NOT #_w1 THEN
       #OUT.F3_ENG := (#OUT.CV_ENG*#FP_RARM.Recipe_Accepted[3])/100.0;
   END_IF;
END_REGION

REGION Network 45: Calculate Feeder 4 Setpoint (t/h)
   IF #FP_EN.Force_Feeder4 THEN #OUT.F4_ENG := #FP_RARM.Force_Values[4]; END_IF;
   #_w1 := #FP_RARM.Recipe_Accepted[4] <= 0.0;
   IF #_w1 THEN #OUT.F4_ENG := 0.0; END_IF;
   IF NOT #FP_EN.Force_Feeder4 AND NOT #_w1 THEN
       #OUT.F4_ENG := (#OUT.CV_ENG*#FP_RARM.Recipe_Accepted[4])/100.0;
   END_IF;
END_REGION

REGION Network 46: Calculate Feeder 5 Setpoint (t/h)
   IF #FP_EN.Force_Feeder5 THEN #OUT.F5_ENG := #FP_RARM.Force_Values[5]; END_IF;
   #_w1 := #FP_RARM.Recipe_Accepted[5] <= 0.0;
   IF #_w1 THEN #OUT.F5_ENG := 0.0; END_IF;
   IF NOT #FP_EN.Force_Feeder5 AND NOT #_w1 THEN
       #OUT.F5_ENG := (#OUT.CV_ENG*#FP_RARM.Recipe_Accepted[5])/100.0;
   END_IF;
END_REGION

REGION Network 47: Calculate Feeder 6 Setpoint (t/h)
   IF #FP_EN.Force_Feeder6 THEN #OUT.F6_ENG := #FP_RARM.Force_Values[6]; END_IF;
   #_w1 := #FP_RARM.Recipe_Accepted[6] <= 0.0;
   IF #_w1 THEN #OUT.F6_ENG := 0.0; END_IF;
   IF NOT #FP_EN.Force_Feeder6 AND NOT #_w1 THEN
       #OUT.F6_ENG := (#OUT.CV_ENG*#FP_RARM.Recipe_Accepted[6])/100.0;
   END_IF;
END_REGION

REGION Network 48: Calculate Feeder 7 Setpoint (t/h)
   IF #FP_EN.Force_Feeder7 THEN #OUT.F7_ENG := #FP_RARM.Force_Values[7]; END_IF;
   #_w1 := #FP_RARM.Recipe_Accepted[7] <= 0.0;
   IF #_w1 THEN #OUT.F7_ENG := 0.0; END_IF;
   IF NOT #FP_EN.Force_Feeder7 AND NOT #_w1 THEN
       #OUT.F7_ENG := (#OUT.CV_ENG*#FP_RARM.Recipe_Accepted[7])/100.0;
   END_IF;
END_REGION

REGION Network 49: Calculate Feeder 8 Setpoint (t/h)
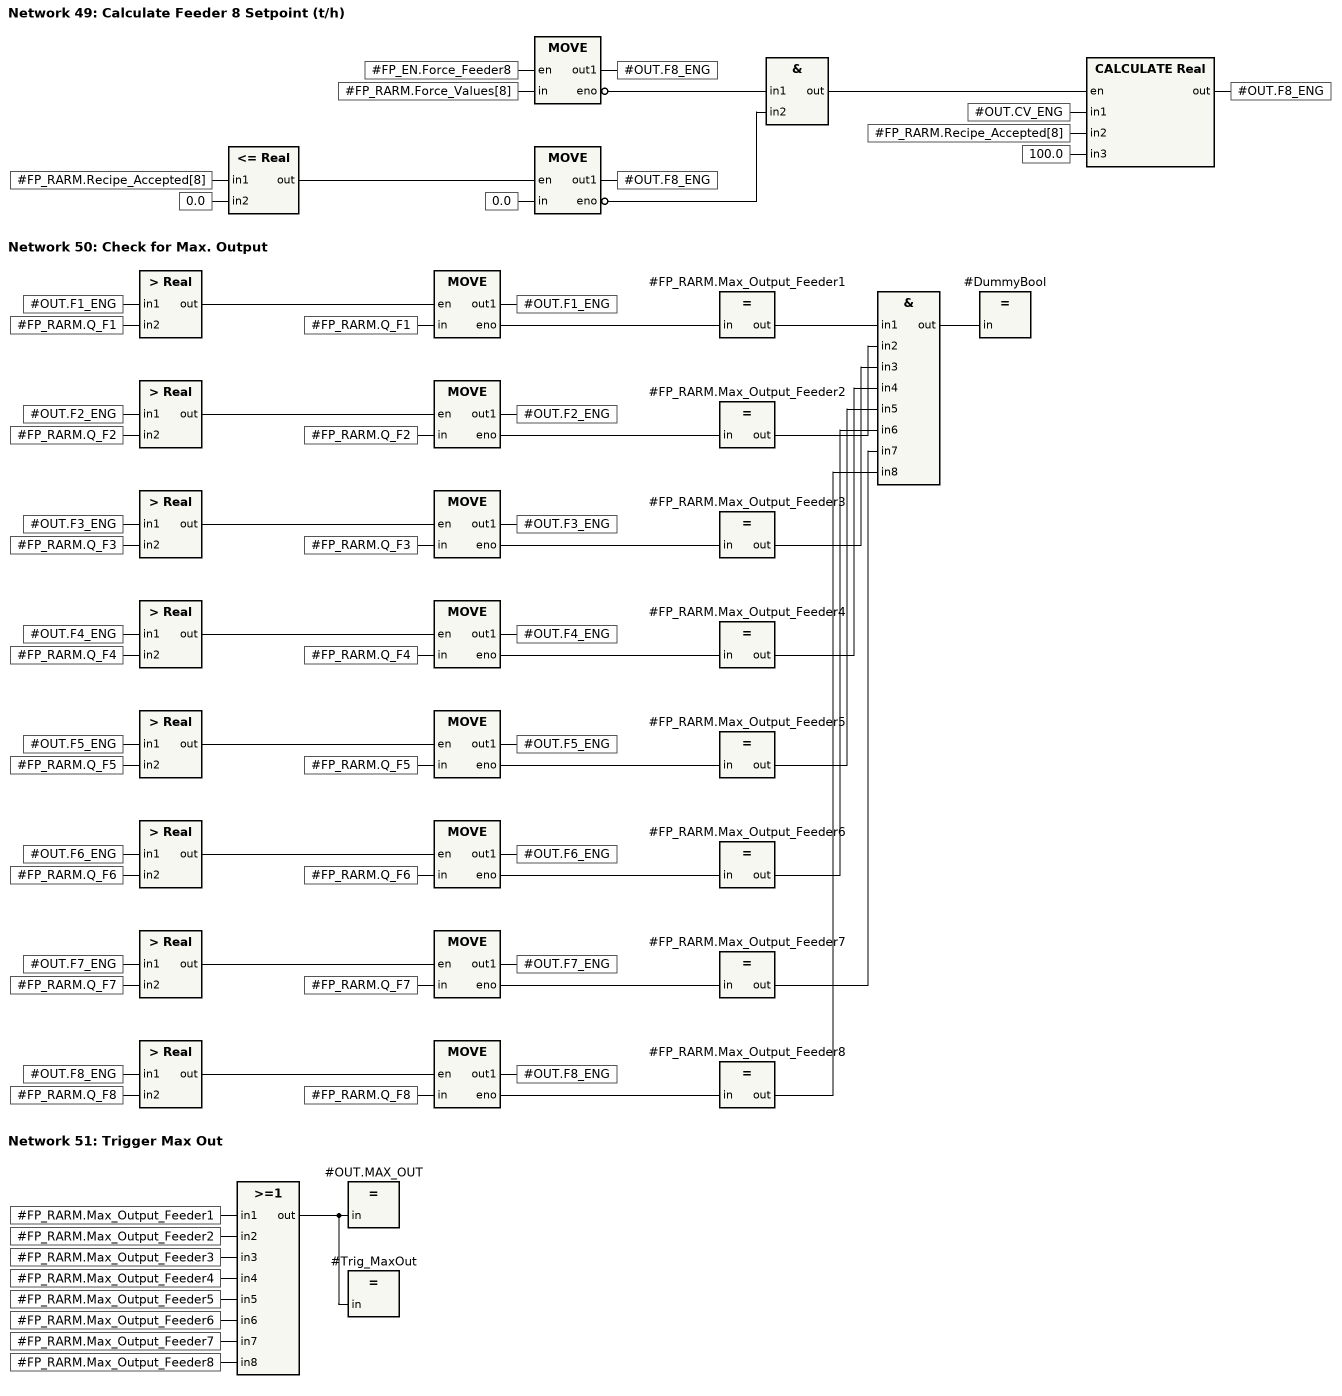
   IF #FP_EN.Force_Feeder8 THEN #OUT.F8_ENG := #FP_RARM.Force_Values[8]; END_IF;
   #_w1 := #FP_RARM.Recipe_Accepted[8] <= 0.0;
   IF #_w1 THEN #OUT.F8_ENG := 0.0; END_IF;
   IF NOT #FP_EN.Force_Feeder8 AND NOT #_w1 THEN
       #OUT.F8_ENG := (#OUT.CV_ENG*#FP_RARM.Recipe_Accepted[8])/100.0;
   END_IF;
END_REGION

REGION Network 50: Check for Max. Output
   #_w1 := #OUT.F1_ENG > #FP_RARM.Q_F1;
   IF #_w1 THEN #OUT.F1_ENG := #FP_RARM.Q_F1; END_IF;
   #FP_RARM.Max_Output_Feeder1 := #_w1;
   #_w2 := #OUT.F2_ENG > #FP_RARM.Q_F2;
   IF #_w2 THEN #OUT.F2_ENG := #FP_RARM.Q_F2; END_IF;
   #FP_RARM.Max_Output_Feeder2 := #_w2;
   #_w3 := #OUT.F3_ENG > #FP_RARM.Q_F3;
   IF #_w3 THEN #OUT.F3_ENG := #FP_RARM.Q_F3; END_IF;
   #FP_RARM.Max_Output_Feeder3 := #_w3;
   #_w4 := #OUT.F4_ENG > #FP_RARM.Q_F4;
   IF #_w4 THEN #OUT.F4_ENG := #FP_RARM.Q_F4; END_IF;
   #FP_RARM.Max_Output_Feeder4 := #_w4;
   #_w5 := #OUT.F5_ENG > #FP_RARM.Q_F5;
   IF #_w5 THEN #OUT.F5_ENG := #FP_RARM.Q_F5; END_IF;
   #FP_RARM.Max_Output_Feeder5 := #_w5;
   #_w6 := #OUT.F6_ENG > #FP_RARM.Q_F6;
   IF #_w6 THEN #OUT.F6_ENG := #FP_RARM.Q_F6; END_IF;
   #FP_RARM.Max_Output_Feeder6 := #_w6;
   #_w7 := #OUT.F7_ENG > #FP_RARM.Q_F7;
   IF #_w7 THEN #OUT.F7_ENG := #FP_RARM.Q_F7; END_IF;
   #FP_RARM.Max_Output_Feeder7 := #_w7;
   #_w8 := #OUT.F8_ENG > #FP_RARM.Q_F8;
   IF #_w8 THEN #OUT.F8_ENG := #FP_RARM.Q_F8; END_IF;
   #FP_RARM.Max_Output_Feeder8 := #_w8;
   #DummyBool := #_w1 AND #_w2 AND #_w3 AND #_w4 AND #_w5 AND #_w6 AND #_w7 AND #_w8;
END_REGION

REGION Network 51: Trigger Max Out
   #OUT.MAX_OUT := #FP_RARM.Max_Output_Feeder1 OR #FP_RARM.Max_Output_Feeder2 OR #FP_RARM.Max_Output_Feeder3 OR #FP_RARM.Max_Output_Feeder4 OR #FP_RARM.Max_Output_Feeder5 OR #FP_RARM.Max_Output_Feeder6 OR #FP_RARM.Max_Output_Feeder7 OR #FP_RARM.Max_Output_Feeder8;
   #Trig_MaxOut := #OUT.MAX_OUT;
END_REGION

REGION Network 52: Calculate Feeder 1 PCT
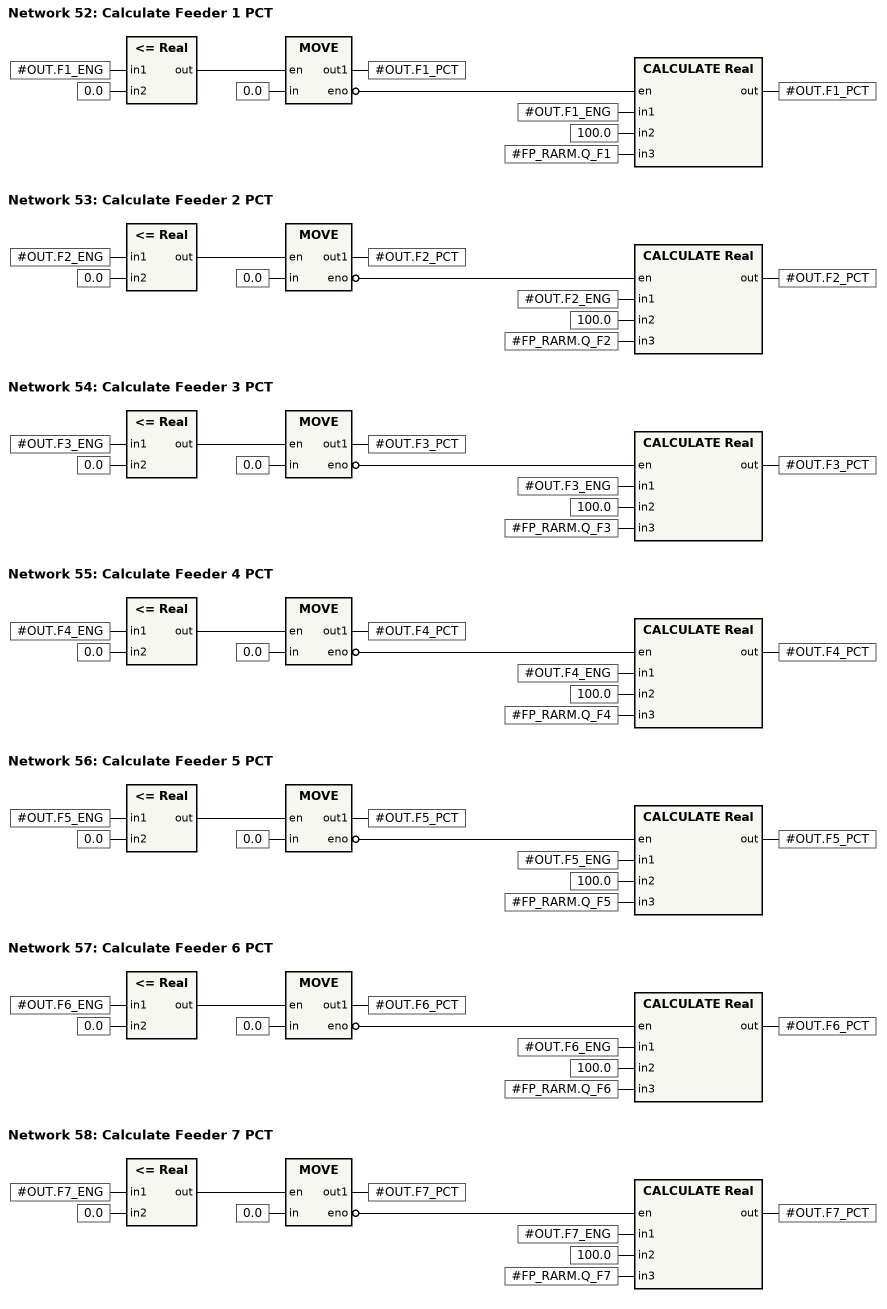
   IF #OUT.F1_ENG <= 0.0 THEN #OUT.F1_PCT := 0.0; END_IF;
   IF NOT (#OUT.F1_ENG <= 0.0) THEN #OUT.F1_PCT := (#OUT.F1_ENG*100.0)/#FP_RARM.Q_F1; END_IF;
END_REGION

REGION Network 53: Calculate Feeder 2 PCT
   IF #OUT.F2_ENG <= 0.0 THEN #OUT.F2_PCT := 0.0; END_IF;
   IF NOT (#OUT.F2_ENG <= 0.0) THEN #OUT.F2_PCT := (#OUT.F2_ENG*100.0)/#FP_RARM.Q_F2; END_IF;
END_REGION

REGION Network 54: Calculate Feeder 3 PCT
   IF #OUT.F3_ENG <= 0.0 THEN #OUT.F3_PCT := 0.0; END_IF;
   IF NOT (#OUT.F3_ENG <= 0.0) THEN #OUT.F3_PCT := (#OUT.F3_ENG*100.0)/#FP_RARM.Q_F3; END_IF;
END_REGION

REGION Network 55: Calculate Feeder 4 PCT
   IF #OUT.F4_ENG <= 0.0 THEN #OUT.F4_PCT := 0.0; END_IF;
   IF NOT (#OUT.F4_ENG <= 0.0) THEN #OUT.F4_PCT := (#OUT.F4_ENG*100.0)/#FP_RARM.Q_F4; END_IF;
END_REGION

REGION Network 56: Calculate Feeder 5 PCT
   IF #OUT.F5_ENG <= 0.0 THEN #OUT.F5_PCT := 0.0; END_IF;
   IF NOT (#OUT.F5_ENG <= 0.0) THEN #OUT.F5_PCT := (#OUT.F5_ENG*100.0)/#FP_RARM.Q_F5; END_IF;
END_REGION

REGION Network 57: Calculate Feeder 6 PCT
   IF #OUT.F6_ENG <= 0.0 THEN #OUT.F6_PCT := 0.0; END_IF;
   IF NOT (#OUT.F6_ENG <= 0.0) THEN #OUT.F6_PCT := (#OUT.F6_ENG*100.0)/#FP_RARM.Q_F6; END_IF;
END_REGION

REGION Network 58: Calculate Feeder 7 PCT
   IF #OUT.F7_ENG <= 0.0 THEN #OUT.F7_PCT := 0.0; END_IF;
   IF NOT (#OUT.F7_ENG <= 0.0) THEN #OUT.F7_PCT := (#OUT.F7_ENG*100.0)/#FP_RARM.Q_F7; END_IF;
END_REGION

REGION Network 59: Calculate Feeder 8 PCT
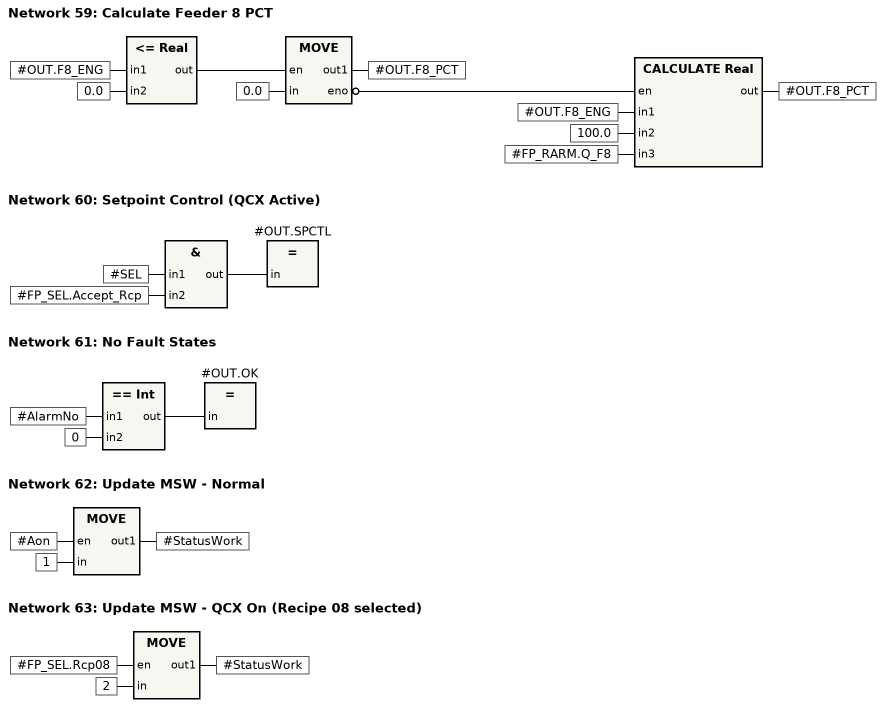
   IF #OUT.F8_ENG <= 0.0 THEN #OUT.F8_PCT := 0.0; END_IF;
   IF NOT (#OUT.F8_ENG <= 0.0) THEN #OUT.F8_PCT := (#OUT.F8_ENG*100.0)/#FP_RARM.Q_F8; END_IF;
END_REGION

REGION Network 60: Setpoint Control (QCX Active)
   #OUT.SPCTL := #SEL AND #FP_SEL.Accept_Rcp;
END_REGION

REGION Network 61: No Fault States
   #OUT.OK := #AlarmNo = 0;
END_REGION

REGION Network 62: Update MSW - Normal
   IF #Aon THEN #StatusWork := 1; END_IF;
END_REGION

REGION Network 63: Update MSW - QCX On (Recipe 08 selected)
   IF #FP_SEL.Rcp08 THEN #StatusWork := 2; END_IF;
END_REGION

REGION Network 64: Update MSW - Not all selected feederes running
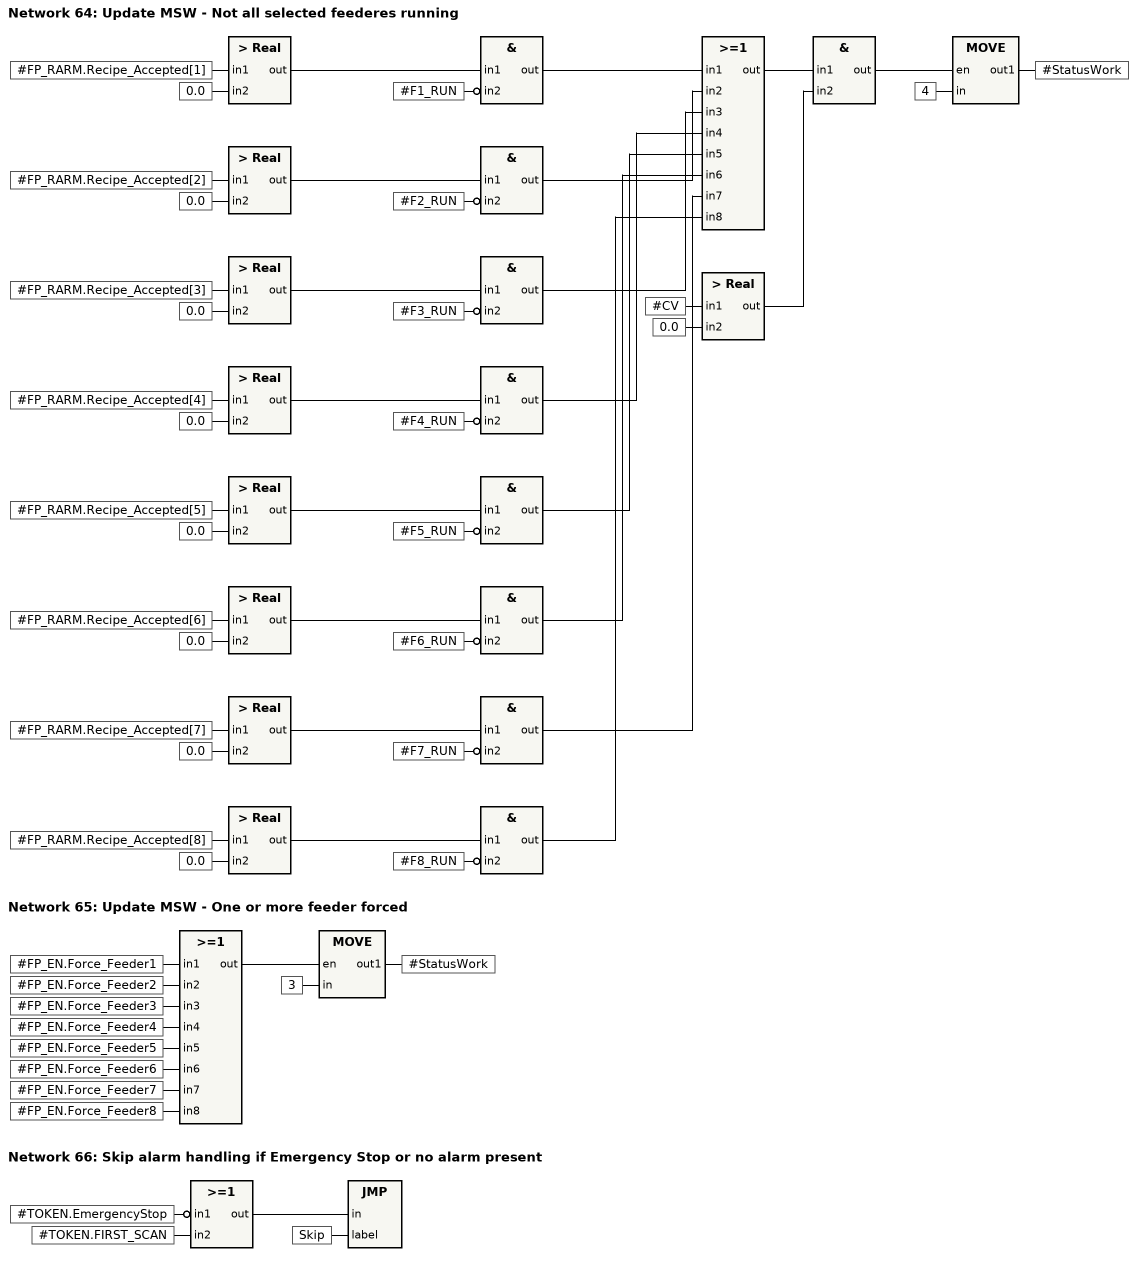
   IF (((#FP_RARM.Recipe_Accepted[1] > 0.0) AND NOT #F1_RUN) OR ((#FP_RARM.Recipe_Accepted[2] > 0.0) AND NOT #F2_RUN) OR ((#FP_RARM.Recipe_Accepted[3] > 0.0) AND NOT #F3_RUN) OR ((#FP_RARM.Recipe_Accepted[4] > 0.0) AND NOT #F4_RUN) OR ((#FP_RARM.Recipe_Accepted[5] > 0.0) AND NOT #F5_RUN) OR ((#FP_RARM.Recipe_Accepted[6] > 0.0) AND NOT #F6_RUN) OR ((#FP_RARM.Recipe_Accepted[7] > 0.0) AND NOT #F7_RUN) OR ((#FP_RARM.Recipe_Accepted[8] > 0.0) AND NOT #F8_RUN)) AND (#CV > 0.0) THEN
       #StatusWork := 4;
   END_IF;
END_REGION

REGION Network 65: Update MSW - One or more feeder forced
   IF #FP_EN.Force_Feeder1 OR #FP_EN.Force_Feeder2 OR #FP_EN.Force_Feeder3 OR #FP_EN.Force_Feeder4 OR #FP_EN.Force_Feeder5 OR #FP_EN.Force_Feeder6 OR #FP_EN.Force_Feeder7 OR #FP_EN.Force_Feeder8 THEN
       #StatusWork := 3;
   END_IF;
END_REGION

REGION Network 66: Skip alarm handling if Emergency Stop or no alarm present
   // Skip = Skip Alarm
   IF NOT #TOKEN.EmergencyStop OR #TOKEN.FIRST_SCAN THEN GOTO Skip; END_IF;
END_REGION

REGION Network 67: Alarm Present
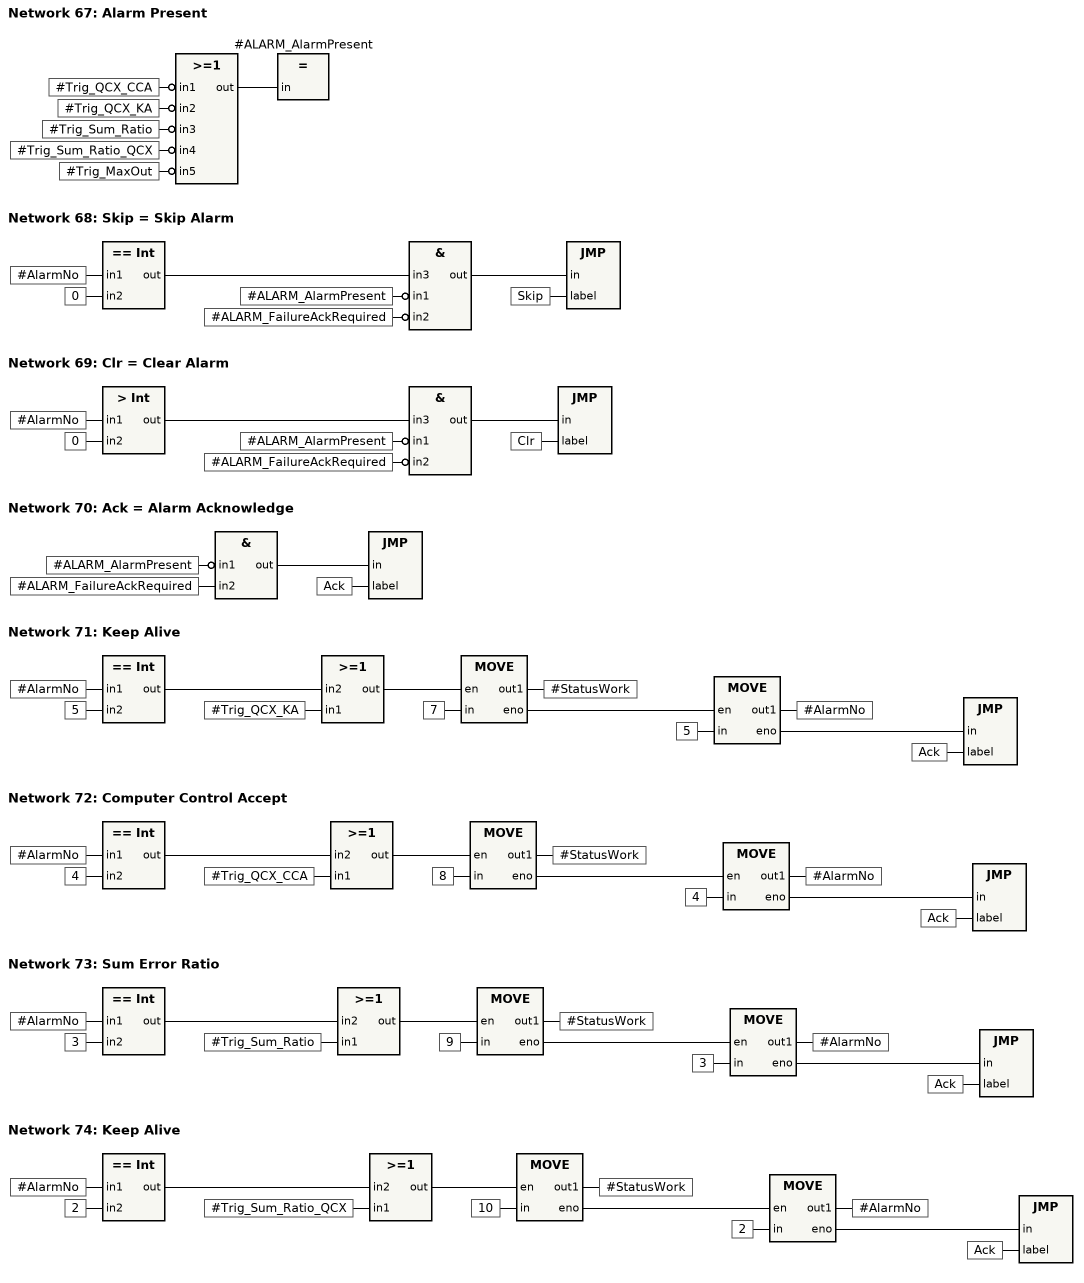
   #ALARM_AlarmPresent := NOT #Trig_QCX_CCA OR NOT #Trig_QCX_KA OR NOT #Trig_Sum_Ratio OR NOT #Trig_Sum_Ratio_QCX OR NOT #Trig_MaxOut;
END_REGION

REGION Network 68: Skip = Skip Alarm
   IF (#AlarmNo = 0) AND NOT #ALARM_AlarmPresent AND NOT #ALARM_FailureAckRequired THEN GOTO Skip; END_IF;
END_REGION

REGION Network 69: Clr = Clear Alarm
   IF (#AlarmNo > 0) AND NOT #ALARM_AlarmPresent AND NOT #ALARM_FailureAckRequired THEN GOTO Clr; END_IF;
END_REGION

REGION Network 70: Ack = Alarm Acknowledge
   IF NOT #ALARM_AlarmPresent AND #ALARM_FailureAckRequired THEN GOTO Ack; END_IF;
END_REGION

REGION Network 71: Keep Alive
   // ENO of a box is taken as its EN; it also drops when the box reports an error
   #_w1 := (#AlarmNo = 5) OR #Trig_QCX_KA;
   IF #_w1 THEN
       #StatusWork := 7;
       #AlarmNo := 5;
       GOTO Ack;
   END_IF;
END_REGION

REGION Network 72: Computer Control Accept
   // ENO of a box is taken as its EN; it also drops when the box reports an error
   #_w1 := (#AlarmNo = 4) OR #Trig_QCX_CCA;
   IF #_w1 THEN
       #StatusWork := 8;
       #AlarmNo := 4;
       GOTO Ack;
   END_IF;
END_REGION

REGION Network 73: Sum Error Ratio
   // ENO of a box is taken as its EN; it also drops when the box reports an error
   #_w1 := (#AlarmNo = 3) OR #Trig_Sum_Ratio;
   IF #_w1 THEN
       #StatusWork := 9;
       #AlarmNo := 3;
       GOTO Ack;
   END_IF;
END_REGION

REGION Network 74: Keep Alive
   // ENO of a box is taken as its EN; it also drops when the box reports an error
   #_w1 := (#AlarmNo = 2) OR #Trig_Sum_Ratio_QCX;
   IF #_w1 THEN
       #StatusWork := 10;
       #AlarmNo := 2;
       GOTO Ack;
   END_IF;
END_REGION

REGION Network 75: Max Output
